KUKA KRL program: EPS_2_251825_SA14_A_20260116064056.src

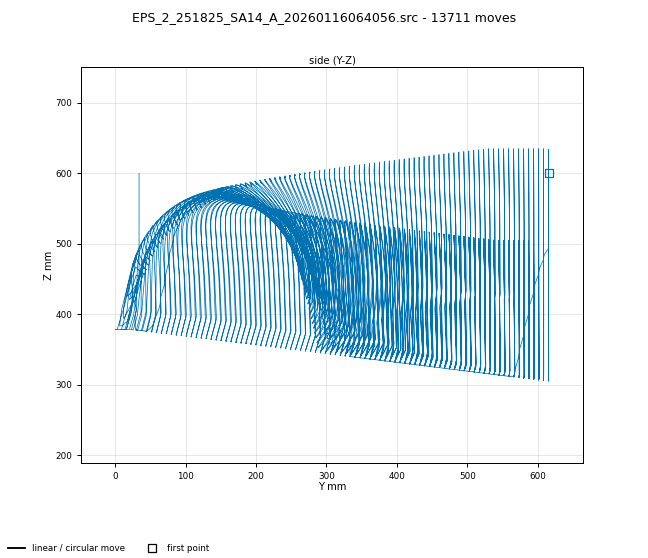
[picture p0: tool path of EPS_2_251825_SA14_A_20260116064056.src, 13711 of 13713 moves have a stored position in this frame; points joined in program order, loops and branches not executed]
&ACCESS RVP
&REL 4
&COMMENT QRS 19112012
&PARAM EDITMASK = *
DEF PART()
EXT BAS (BAS_COMMAND :IN,REAL :IN )
INT I
BAS (#INITMOV,0 )

;KUKA QRS Post kuka4.cps  Date:22-06-2017 !

File_ID=2976

QRS_PRE_INIT()

;Init var - Until changes are made in qrs_pre_init
Outlet_Square_prg=0
Inlet_1_Square_prg=0
Inlet_2_Square_prg=0
Inlet_3_Square_prg=0
Inlet_4_Square_prg=0
Inlet_5_Square_prg=0

Outlet_1={X 0.000, Y 530.070, Z 534.500, B 0.000, E1 0.000 }
Inlet_1={X 0.000, Y 539.340, Z 404.500, B 0.000, E1 92.000 }
Inlet_2={X 0.000, Y 539.340, Z 404.500, B 0.000, E1 262.000 }
Outlet_1_type=201
Inlet_1_type=201
Inlet_2_type=201
;QRS#1=Sidecore dimensions
;QRS#2=200-8" PVC SDR 35
;QRS#3=200-8" PVC SDR 35
;QRS#4=200-8" PVC SDR 35
;QRS#5=
;QRS#6=
;QRS#7=
;QRS#8=
;QRS#9=12-08 PSX
;QRS#10=12-08 PSX
;QRS#11=12-08 PSX
;QRS#12=
;QRS#13=
;QRS#14=
;QRS#15=
;QRS#16=1220x127x914 3'
;QRS#17=EPS Height
;QRS#18=635
;QRS#19=*
;QRS#20= UPDATED VERSION 22-06-2017
;QRS#21=*
Outlet_Square=0100
Inlet_1_Square=0100
Inlet_2_Square=0100
Inlet_3_Square=0
Inlet_4_Square=0
Inlet_5_Square=0
Mill_Square=1
Outlet_Square_Prg=204
Inlet_1_Square_prg=204
Inlet_2_Square_prg=204

QRS_INIT()

$ADVANCE=5

; T1
PTP {E1 173.528,E2 173.528}
PTP {X 0,Y 615.502,A -85,B 0,C 180,E1 173.528,E2 173.528,E3 0,E4 0,E5 0,E6 0}
QRS_SPEED_INIT()
LIN {X 0,Y 615.502,Z 600,A -85,B 0,C 180,E1 173.528,E2 173.528,E3 0,E4 0,E5 0,E6 0} C_VEL
LIN {X 0,Y 615.502,Z 506.059,A -85,B 0,C 180,E1 173.528,E2 173.528} C_VEL
LIN {X 0,Y 615.502,Z 496.473,A -85,B 0,C 180,E1 173.528,E2 173.528} C_VEL
LIN {X 0,Y 615.497,Z 494.64,A -85,B 0,C 180,E1 173.417,E2 173.417} C_VEL
LIN {X 0,Y 615.496,Z 489.786,A -85,B 0,C 180,E1 172.455,E2 172.455} C_VEL
LIN {X 0,Y 615.498,Z 483.532,A -85,B 0,C 180,E1 171.464,E2 171.464} C_VEL
LIN {X 0,Y 615.498,Z 475.676,A -85,B 0,C 180,E1 170.47,E2 170.47} C_VEL
LIN {X 0,Y 615.498,Z 465.867,A -85,B 0,C 180,E1 169.474,E2 169.474} C_VEL
LIN {X 0,Y 615.499,Z 455.563,A -85,B 0,C 180,E1 168.641,E2 168.641} C_VEL
LIN {X 0,Y 615.479,Z 445.348,A -85,B 0,C 180,E1 167.972,E2 167.972} C_VEL
LIN {X 0,Y 615.497,Z 434.148,A -85,B 0,C 180,E1 167.387,E2 167.387} C_VEL
LIN {X 0,Y 615.49,Z 421.521,A -85,B 0,C 180,E1 166.883,E2 166.883} C_VEL
LIN {X 0,Y 615.487,Z 409.783,A -85,B 0,C 180,E1 166.547,E2 166.547} C_VEL
LIN {X 0,Y 615.473,Z 395.857,A -85,B 0,C 180,E1 166.294,E2 166.294} C_VEL
LIN {X 0,Y 615.498,Z 304.699,A -85,B 0,C 180,E1 165.219,E2 165.219} C_VEL
LIN {X 0,Y 615.493,Z 304.685,A -85,B 0,C 180,E1 162.73,E2 162.73} C_VEL
LIN {X 0,Y 615.461,Z 304.691,A -85,B 0,C 180,E1 159.967,E2 159.967} C_VEL
LIN {X 0,Y 615.471,Z 304.695,A -85,B 0,C 180,E1 157.658,E2 157.658} C_VEL
LIN {X 0,Y 615.486,Z 304.691,A -85,B 0,C 180,E1 155.009,E2 155.009} C_VEL
LIN {X 0,Y 615.486,Z 304.687,A -85,B 0,C 180,E1 152.823,E2 152.823} C_VEL
LIN {X 0,Y 615.466,Z 304.688,A -85,B 0,C 180,E1 150.209,E2 150.209} C_VEL
LIN {X 0,Y 615.483,Z 304.7,A -85,B 0,C 180,E1 147.543,E2 147.543} C_VEL
LIN {X 0,Y 615.488,Z 304.693,A -85,B 0,C 180,E1 145.185,E2 145.185} C_VEL
LIN {X 0,Y 615.49,Z 304.683,A -85,B 0,C 180,E1 142.758,E2 142.758} C_VEL
LIN {X 0,Y 615.467,Z 304.694,A -85,B 0,C 180,E1 139.914,E2 139.914} C_VEL
LIN {X 0,Y 615.487,Z 304.698,A -85,B 0,C 180,E1 137.647,E2 137.647} C_VEL
LIN {X 0,Y 615.483,Z 304.686,A -85,B 0,C 180,E1 134.932,E2 134.932} C_VEL
LIN {X 0,Y 615.467,Z 304.692,A -85,B 0,C 180,E1 132.079,E2 132.079} C_VEL
LIN {X 0,Y 615.484,Z 304.698,A -85,B 0,C 180,E1 129.751,E2 129.751} C_VEL
LIN {X 0,Y 615.484,Z 304.685,A -85,B 0,C 180,E1 126.937,E2 126.937} C_VEL
LIN {X 0,Y 615.49,Z 304.682,A -85,B 0,C 180,E1 124.702,E2 124.702} C_VEL
LIN {X 0,Y 615.47,Z 304.689,A -85,B 0,C 180,E1 122.329,E2 122.329} C_VEL
LIN {X 0,Y 615.489,Z 304.699,A -85,B 0,C 180,E1 119.796,E2 119.796} C_VEL
LIN {X 0,Y 615.487,Z 304.684,A -85,B 0,C 180,E1 117.046,E2 117.046} C_VEL
LIN {X 0,Y 615.489,Z 304.683,A -85,B 0,C 180,E1 114.992,E2 114.992} C_VEL
LIN {X 0,Y 615.475,Z 304.693,A -85,B 0,C 180,E1 112.137,E2 112.137} C_VEL
LIN {X 0,Y 615.48,Z 304.69,A -85,B 0,C 180,E1 109.338,E2 109.338} C_VEL
LIN {X 0,Y 615.478,Z 304.686,A -85,B 0,C 180,E1 106.587,E2 106.587} C_VEL
LIN {X 0,Y 615.497,Z 304.7,A -85,B 0,C 180,E1 103.874,E2 103.874} C_VEL
LIN {X 0,Y 615.486,Z 304.683,A -85,B 0,C 180,E1 100.889,E2 100.889} C_VEL
LIN {X 0,Y 615.476,Z 304.688,A -85,B 0,C 180,E1 98.537,E2 98.537} C_VEL
LIN {X 0,Y 615.496,Z 304.7,A -85,B 0,C 180,E1 95.898,E2 95.898} C_VEL
LIN {X 0,Y 615.482,Z 304.686,A -85,B 0,C 180,E1 93.273,E2 93.273} C_VEL
LIN {X 0,Y 615.479,Z 304.686,A -85,B 0,C 180,E1 90.654,E2 90.654} C_VEL
LIN {X 0,Y 615.496,Z 304.7,A -85,B 0,C 180,E1 88.037,E2 88.037} C_VEL
LIN {X 0,Y 615.477,Z 304.688,A -85,B 0,C 180,E1 85.415,E2 85.415} C_VEL
LIN {X 0,Y 615.483,Z 304.685,A -85,B 0,C 180,E1 82.784,E2 82.784} C_VEL
LIN {X 0,Y 615.493,Z 304.699,A -85,B 0,C 180,E1 80.138,E2 80.138} C_VEL
LIN {X 0,Y 615.477,Z 304.687,A -85,B 0,C 180,E1 77.469,E2 77.469} C_VEL
LIN {X 0,Y 615.482,Z 304.686,A -85,B 0,C 180,E1 74.774,E2 74.774} C_VEL
LIN {X 0,Y 615.49,Z 304.698,A -85,B 0,C 180,E1 72.043,E2 72.043} C_VEL
LIN {X 0,Y 615.487,Z 304.682,A -85,B 0,C 180,E1 69.269,E2 69.269} C_VEL
LIN {X 0,Y 615.485,Z 304.695,A -85,B 0,C 180,E1 66.443,E2 66.443} C_VEL
LIN {X 0,Y 615.496,Z 304.699,A -85,B 0,C 180,E1 64.284,E2 64.284} C_VEL
LIN {X 0,Y 615.482,Z 304.683,A -85,B 0,C 180,E1 61.341,E2 61.341} C_VEL
LIN {X 0,Y 615.485,Z 304.686,A -85,B 0,C 180,E1 58.914,E2 58.914} C_VEL
LIN {X 0,Y 615.476,Z 304.694,A -85,B 0,C 180,E1 55.977,E2 55.977} C_VEL
LIN {X 0,Y 615.473,Z 304.687,A -85,B 0,C 180,E1 53.574,E2 53.574} C_VEL
LIN {X 0,Y 615.485,Z 304.686,A -85,B 0,C 180,E1 50.938,E2 50.938} C_VEL
LIN {X 0,Y 615.489,Z 304.697,A -85,B 0,C 180,E1 48.526,E2 48.526} C_VEL
LIN {X 0,Y 615.469,Z 304.69,A -85,B 0,C 180,E1 45.848,E2 45.848} C_VEL
LIN {X 0,Y 615.488,Z 304.685,A -85,B 0,C 180,E1 43.047,E2 43.047} C_VEL
LIN {X 0,Y 615.49,Z 304.697,A -85,B 0,C 180,E1 40.606,E2 40.606} C_VEL
LIN {X 0,Y 615.469,Z 304.692,A -85,B 0,C 180,E1 38.009,E2 38.009} C_VEL
LIN {X 0,Y 615.473,Z 304.686,A -85,B 0,C 180,E1 35.616,E2 35.616} C_VEL
LIN {X 0,Y 615.49,Z 304.683,A -85,B 0,C 180,E1 33.236,E2 33.236} C_VEL
LIN {X 0,Y 615.486,Z 304.691,A -85,B 0,C 180,E1 30.919,E2 30.919} C_VEL
LIN {X 0,Y 615.485,Z 304.699,A -85,B 0,C 180,E1 28.449,E2 28.449} C_VEL
LIN {X 0,Y 615.48,Z 304.684,A -85,B 0,C 180,E1 25.566,E2 25.566} C_VEL
LIN {X 0,Y 615.486,Z 304.696,A -85,B 0,C 180,E1 22.844,E2 22.844} C_VEL
LIN {X 0,Y 615.487,Z 304.702,A -85,B 0,C 180,E1 20.686,E2 20.686} C_VEL
LIN {X 0,Y 615.486,Z 401.466,A -85,B 0,C 180,E1 19.533,E2 19.533} C_VEL
LIN {X 0,Y 615.49,Z 414.153,A -85,B 0,C 180,E1 19.251,E2 19.251} C_VEL
LIN {X 0,Y 615.49,Z 427.253,A -85,B 0,C 180,E1 18.818,E2 18.818} C_VEL
LIN {X 0,Y 615.491,Z 439.133,A -85,B 0,C 180,E1 18.281,E2 18.281} C_VEL
LIN {X 0,Y 615.485,Z 450.58,A -85,B 0,C 180,E1 17.613,E2 17.613} C_VEL
LIN {X 0,Y 615.497,Z 461.144,A -85,B 0,C 180,E1 16.842,E2 16.842} C_VEL
LIN {X 0,Y 615.499,Z 470.075,A -85,B 0,C 180,E1 16.036,E2 16.036} C_VEL
LIN {X 0,Y 615.497,Z 478.904,A -85,B 0,C 180,E1 15.056,E2 15.056} C_VEL
LIN {X 0,Y 615.498,Z 485.954,A -85,B 0,C 180,E1 14.088,E2 14.088} C_VEL
LIN {X 0,Y 615.499,Z 491.179,A -85,B 0,C 180,E1 13.201,E2 13.201} C_VEL
LIN {X 0,Y 615.495,Z 495.923,A -85,B 0,C 180,E1 12.195,E2 12.195} C_VEL
LIN {X 0,Y 615.496,Z 499.511,A -85,B 0,C 180,E1 11.193,E2 11.193} C_VEL
LIN {X 0,Y 615.497,Z 501.344,A -85,B 0,C 180,E1 10.526,E2 10.526} C_VEL
LIN {X 0,Y 615.495,Z 502.702,A -85,B 0,C 180,E1 9.862,E2 9.862} C_VEL
LIN {X 0,Y 615.496,Z 504.225,A -85,B 0,C 180,E1 8.536,E2 8.536} C_VEL
LIN {X 0,Y 615.495,Z 504.376,A -85,B 0,C 180,E1 7.875,E2 7.875} C_VEL
LIN {X 0,Y 615.497,Z 503.473,A -85,B 0,C 180,E1 6.556,E2 6.556} C_VEL
LIN {X 0,Y 615.499,Z 502.449,A -85,B 0,C 180,E1 5.898,E2 5.898} C_VEL
LIN {X 0,Y 615.495,Z 500.977,A -85,B 0,C 180,E1 5.241,E2 5.241} C_VEL
LIN {X 0,Y 615.496,Z 497.999,A -85,B 0,C 180,E1 4.256,E2 4.256} C_VEL
LIN {X 0,Y 615.496,Z 493.997,A -85,B 0,C 180,E1 3.273,E2 3.273} C_VEL
LIN {X 0,Y 615.496,Z 487.85,A -85,B 0,C 180,E1 2.126,E2 2.126} C_VEL
LIN {X 0,Y 615.498,Z 481.175,A -85,B 0,C 180,E1 1.145,E2 1.145} C_VEL
LIN {X 0,Y 615.498,Z 472.909,A -85,B 0,C 180,E1 0.163,E2 0.163} C_VEL
LIN {X 0,Y 615.498,Z 464.406,A -85,B 0,C 180,E1 -0.655,E2 -0.655} C_VEL
LIN {X 0,Y 615.493,Z 453.986,A -85,B 0,C 180,E1 -1.472,E2 -1.472} C_VEL
LIN {X 0,Y 615.476,Z 443.668,A -85,B 0,C 180,E1 -2.127,E2 -2.127} C_VEL
LIN {X 0,Y 615.49,Z 432.239,A -85,B 0,C 180,E1 -2.7,E2 -2.7} C_VEL
LIN {X 0,Y 615.452,Z 420.503,A -85,B 0,C 180,E1 -3.151,E2 -3.151} C_VEL
LIN {X 0,Y 615.434,Z 408.729,A -85,B 0,C 180,E1 -3.478,E2 -3.478} C_VEL
LIN {X 0,Y 615.432,Z 396.068,A -85,B 0,C 180,E1 -3.704,E2 -3.704} C_VEL
LIN {X 0,Y 615.484,Z 304.701,A -85,B 0,C 180,E1 -4.79,E2 -4.79} C_VEL
LIN {X 0,Y 615.438,Z 304.698,A -85,B 0,C 180,E1 -7.217,E2 -7.217} C_VEL
LIN {X 0,Y 615.432,Z 304.699,A -85,B 0,C 180,E1 -9.2,E2 -9.2} C_VEL
LIN {X 0,Y 615.431,Z 304.699,A -85,B 0,C 180,E1 -11.194,E2 -11.194} C_VEL
LIN {X 0,Y 615.426,Z 304.699,A -85,B 0,C 180,E1 -13.203,E2 -13.203} C_VEL
LIN {X 0,Y 615.421,Z 304.699,A -85,B 0,C 180,E1 -15.228,E2 -15.228} C_VEL
LIN {X 0,Y 615.415,Z 304.7,A -85,B 0,C 180,E1 -17.273,E2 -17.273} C_VEL
LIN {X 0,Y 615.411,Z 304.7,A -85,B 0,C 180,E1 -19.341,E2 -19.341} C_VEL
LIN {X 0,Y 615.412,Z 304.7,A -85,B 0,C 180,E1 -21.435,E2 -21.435} C_VEL
LIN {X 0,Y 615.456,Z 304.7,A -85,B 0,C 180,E1 -24.001,E2 -24.001} C_VEL
LIN {X 0,Y 615.486,Z 304.696,A -85,B 0,C 180,E1 -26.445,E2 -26.445} C_VEL
LIN {X 0,Y 615.456,Z 304.696,A -85,B 0,C 180,E1 -28.66,E2 -28.66} C_VEL
LIN {X 0,Y 615.428,Z 304.696,A -85,B 0,C 180,E1 -31.076,E2 -31.076} C_VEL
LIN {X 0,Y 615.428,Z 304.697,A -85,B 0,C 180,E1 -33.24,E2 -33.24} C_VEL
LIN {X 0,Y 615.471,Z 304.699,A -85,B 0,C 180,E1 -35.831,E2 -35.831} C_VEL
LIN {X 0,Y 615.49,Z 304.699,A -85,B 0,C 180,E1 -38.069,E2 -38.069} C_VEL
LIN {X 0,Y 615.46,Z 304.691,A -85,B 0,C 180,E1 -40.609,E2 -40.609} C_VEL
LIN {X 0,Y 615.441,Z 304.694,A -85,B 0,C 180,E1 -43.042,E2 -43.042} C_VEL
LIN {X 0,Y 615.443,Z 304.694,A -85,B 0,C 180,E1 -45.073,E2 -45.073} C_VEL
LIN {X 0,Y 615.483,Z 304.699,A -85,B 0,C 180,E1 -47.646,E2 -47.646} C_VEL
LIN {X 0,Y 615.493,Z 304.686,A -85,B 0,C 180,E1 -50.25,E2 -50.25} C_VEL
LIN {X 0,Y 615.454,Z 304.69,A -85,B 0,C 180,E1 -52.755,E2 -52.755} C_VEL
LIN {X 0,Y 615.469,Z 304.697,A -85,B 0,C 180,E1 -55.302,E2 -55.302} C_VEL
LIN {X 0,Y 615.482,Z 304.685,A -85,B 0,C 180,E1 -58.314,E2 -58.314} C_VEL
LIN {X 0,Y 615.465,Z 304.688,A -85,B 0,C 180,E1 -60.592,E2 -60.592} C_VEL
LIN {X 0,Y 615.464,Z 304.693,A -85,B 0,C 180,E1 -62.96,E2 -62.96} C_VEL
LIN {X 0,Y 615.467,Z 304.836,A -85,B 0,C 180,E1 -64.578,E2 -64.578} C_VEL
LIN {X 0,Y 615.488,Z 329.133,A -85,B 0,C 180,E1 -67.281,E2 -67.281} C_VEL
LIN {X 0,Y 615.496,Z 355.374,A -85,B 0,C 180,E1 -70.141,E2 -70.141} C_VEL
LIN {X 0,Y 615.493,Z 382.737,A -85,B 0,C 180,E1 -73.072,E2 -73.072} C_VEL
LIN {X 0,Y 615.499,Z 411.083,A -85,B 0,C 180,E1 -76.064,E2 -76.064} C_VEL
LIN {X 0,Y 615.498,Z 421.301,A -85,B 0,C 180,E1 -77.114,E2 -77.114} C_VEL
LIN {X 0,Y 615.479,Z 530.821,A -85,B 0,C 180,E1 -78.41,E2 -78.41} C_VEL
LIN {X 0,Y 615.478,Z 543.339,A -85,B 0,C 180,E1 -78.681,E2 -78.681} C_VEL
LIN {X 0,Y 615.491,Z 556.57,A -85,B 0,C 180,E1 -79.111,E2 -79.111} C_VEL
LIN {X 0,Y 615.478,Z 568.475,A -85,B 0,C 180,E1 -79.639,E2 -79.639} C_VEL
LIN {X 0,Y 615.487,Z 579.992,A -85,B 0,C 180,E1 -80.304,E2 -80.304} C_VEL
LIN {X 0,Y 615.499,Z 590.339,A -85,B 0,C 180,E1 -81.05,E2 -81.05} C_VEL
LIN {X 0,Y 615.497,Z 598.81,A -85,B 0,C 180,E1 -81.794,E2 -81.794} C_VEL
LIN {X 0,Y 615.498,Z 606.605,A -85,B 0,C 180,E1 -82.619,E2 -82.619} C_VEL
LIN {X 0,Y 615.496,Z 614.202,A -85,B 0,C 180,E1 -83.608,E2 -83.608} C_VEL
LIN {X 0,Y 615.498,Z 621.204,A -85,B 0,C 180,E1 -84.759,E2 -84.759} C_VEL
LIN {X 0,Y 615.493,Z 625.851,A -85,B 0,C 180,E1 -85.743,E2 -85.743} C_VEL
LIN {X 0,Y 615.495,Z 629.398,A -85,B 0,C 180,E1 -86.727,E2 -86.727} C_VEL
LIN {X 0,Y 615.497,Z 631.233,A -85,B 0,C 180,E1 -87.382,E2 -87.382} C_VEL
LIN {X 0,Y 615.497,Z 632.608,A -85,B 0,C 180,E1 -88.037,E2 -88.037} C_VEL
LIN {X 0,Y 615.496,Z 634.173,A -85,B 0,C 180,E1 -89.346,E2 -89.346} C_VEL
LIN {X 0,Y 615.494,Z 634.389,A -85,B 0,C 180,E1 -90,E2 -90} C_VEL
LIN {X 0,Y 615.496,Z 633.58,A -85,B 0,C 180,E1 -91.308,E2 -91.308} C_VEL
LIN {X 0,Y 615.497,Z 632.608,A -85,B 0,C 180,E1 -91.963,E2 -91.963} C_VEL
LIN {X 0,Y 615.497,Z 631.233,A -85,B 0,C 180,E1 -92.618,E2 -92.618} C_VEL
LIN {X 0,Y 615.496,Z 628.35,A -85,B 0,C 180,E1 -93.601,E2 -93.601} C_VEL
LIN {X 0,Y 615.498,Z 624.442,A -85,B 0,C 180,E1 -94.584,E2 -94.584} C_VEL
LIN {X 0,Y 615.499,Z 619.405,A -85,B 0,C 180,E1 -95.57,E2 -95.57} C_VEL
LIN {X 0,Y 615.497,Z 612.87,A -85,B 0,C 180,E1 -96.583,E2 -96.583} C_VEL
LIN {X 0,Y 615.497,Z 605.134,A -85,B 0,C 180,E1 -97.545,E2 -97.545} C_VEL
LIN {X 0,Y 615.498,Z 597.045,A -85,B 0,C 180,E1 -98.371,E2 -98.371} C_VEL
LIN {X 0,Y 615.499,Z 587.168,A -85,B 0,C 180,E1 -99.199,E2 -99.199} C_VEL
LIN {X 0,Y 615.488,Z 575.982,A -85,B 0,C 180,E1 -99.945,E2 -99.945} C_VEL
LIN {X 0,Y 615.481,Z 565.024,A -85,B 0,C 180,E1 -100.527,E2 -100.527} C_VEL
LIN {X 0,Y 615.49,Z 552.45,A -85,B 0,C 180,E1 -101.041,E2 -101.041} C_VEL
LIN {X 0,Y 615.477,Z 540.068,A -85,B 0,C 180,E1 -101.402,E2 -101.402} C_VEL
LIN {X 0,Y 615.481,Z 526.47,A -85,B 0,C 180,E1 -101.652,E2 -101.652} C_VEL
LIN {X 0,Y 615.499,Z 420.901,A -85,B 0,C 180,E1 -102.907,E2 -102.907} C_VEL
LIN {X 0,Y 615.486,Z 393.999,A -85,B 0,C 180,E1 -105.735,E2 -105.735} C_VEL
LIN {X 0,Y 615.477,Z 368.567,A -85,B 0,C 180,E1 -108.441,E2 -108.441} C_VEL
LIN {X 0,Y 615.498,Z 344.101,A -85,B 0,C 180,E1 -111.081,E2 -111.081} C_VEL
LIN {X 0,Y 615.487,Z 318.499,A -85,B 0,C 180,E1 -113.895,E2 -113.895} C_VEL
LIN {X 0,Y 615.468,Z 304.687,A -85,B 0,C 180,E1 -115.458,E2 -115.458} C_VEL
LIN {X 0,Y 615.493,Z 304.699,A -85,B 0,C 180,E1 -118.451,E2 -118.451} C_VEL
LIN {X 0,Y 615.457,Z 304.693,A -85,B 0,C 180,E1 -121.081,E2 -121.081} C_VEL
LIN {X 0,Y 615.471,Z 304.687,A -85,B 0,C 180,E1 -123.531,E2 -123.531} C_VEL
LIN {X 0,Y 615.483,Z 304.701,A -85,B 0,C 180,E1 -126.425,E2 -126.425} C_VEL
LIN {X 0,Y 615.449,Z 304.692,A -85,B 0,C 180,E1 -129.057,E2 -129.057} C_VEL
LIN {X 0,Y 615.467,Z 304.689,A -85,B 0,C 180,E1 -131.476,E2 -131.476} C_VEL
LIN {X 0,Y 615.496,Z 304.7,A -85,B 0,C 180,E1 -134.149,E2 -134.149} C_VEL
LIN {X 0,Y 615.442,Z 304.695,A -85,B 0,C 180,E1 -136.751,E2 -136.751} C_VEL
LIN {X 0,Y 615.437,Z 304.695,A -85,B 0,C 180,E1 -138.911,E2 -138.911} C_VEL
LIN {X 0,Y 615.439,Z 304.694,A -85,B 0,C 180,E1 -141.092,E2 -141.092} C_VEL
LIN {X 0,Y 615.479,Z 304.693,A -85,B 0,C 180,E1 -143.574,E2 -143.574} C_VEL
LIN {X 0,Y 615.436,Z 304.698,A -85,B 0,C 180,E1 -146.473,E2 -146.473} C_VEL
LIN {X 0,Y 615.443,Z 304.699,A -85,B 0,C 180,E1 -148.312,E2 -148.312} C_VEL
LIN {X 0,Y 615.423,Z 304.698,A -85,B 0,C 180,E1 -150.59,E2 -150.59} C_VEL
LIN {X 0,Y 615.424,Z 304.698,A -85,B 0,C 180,E1 -152.967,E2 -152.967} C_VEL
LIN {X 0,Y 615.482,Z 304.702,A -85,B 0,C 180,E1 -155.727,E2 -155.727} C_VEL
LIN {X 0,Y 615.462,Z 304.701,A -85,B 0,C 180,E1 -157.862,E2 -157.862} C_VEL
LIN {X 0,Y 615.448,Z 304.699,A -85,B 0,C 180,E1 -159.966,E2 -159.966} C_VEL
LIN {X 0,Y 615.441,Z 304.698,A -85,B 0,C 180,E1 -162.041,E2 -162.041} C_VEL
LIN {X 0,Y 615.436,Z 304.697,A -85,B 0,C 180,E1 -164.093,E2 -164.093} C_VEL
LIN {X 0,Y 615.435,Z 304.697,A -85,B 0,C 180,E1 -166.124,E2 -166.124} C_VEL
LIN {X 0,Y 615.435,Z 304.696,A -85,B 0,C 180,E1 -168.138,E2 -168.138} C_VEL
LIN {X 0,Y 615.482,Z 304.701,A -85,B 0,C 180,E1 -169.299,E2 -169.299} C_VEL
LIN {X 0,Y 615.427,Z 401.605,A -85,B 0,C 180,E1 -170.468,E2 -170.468} C_VEL
LIN {X 0,Y 615.437,Z 414.547,A -85,B 0,C 180,E1 -170.759,E2 -170.759} C_VEL
LIN {X 0,Y 615.471,Z 427.039,A -85,B 0,C 180,E1 -171.173,E2 -171.173} C_VEL
LIN {X 0,Y 615.487,Z 438.981,A -85,B 0,C 180,E1 -171.711,E2 -171.711} C_VEL
LIN {X 0,Y 615.486,Z 450.346,A -85,B 0,C 180,E1 -172.372,E2 -172.372} C_VEL
LIN {X 0,Y 615.498,Z 460.41,A -85,B 0,C 180,E1 -173.1,E2 -173.1} C_VEL
LIN {X 0,Y 615.497,Z 469.813,A -85,B 0,C 180,E1 -173.937,E2 -173.937} C_VEL
LIN {X 0,Y 615.496,Z 478.73,A -85,B 0,C 180,E1 -174.923,E2 -174.923} C_VEL
LIN {X 0,Y 615.497,Z 485.922,A -85,B 0,C 180,E1 -175.907,E2 -175.907} C_VEL
LIN {X 0,Y 615.497,Z 490.782,A -85,B 0,C 180,E1 -176.727,E2 -176.727} C_VEL
LIN {X 0,Y 615.496,Z 495.51,A -85,B 0,C 180,E1 -177.709,E2 -177.709} C_VEL
LIN {X 0,Y 615.497,Z 499.139,A -85,B 0,C 180,E1 -178.691,E2 -178.691} C_VEL
LIN {X 0,Y 615.495,Z 501.016,A -85,B 0,C 180,E1 -179.345,E2 -179.345} C_VEL
LIN {X 0,Y 615.494,Z 502.471,A -85,B 0,C 180,E1 -180,E2 -180} C_VEL
LIN {X 0,Y 615.495,Z 504.115,A -85,B 0,C 180,E1 -181.308,E2 -181.308} C_VEL
LIN {X 0,Y 615.497,Z 504.374,A -85,B 0,C 180,E1 -181.963,E2 -181.963} C_VEL
LIN {X 0,Y 615.497,Z 504.231,A -85,B 0,C 180,E1 -182.618,E2 -182.618} C_VEL
LIN {X 0,Y 615.496,Z 502.741,A -85,B 0,C 180,E1 -183.928,E2 -183.928} C_VEL
LIN {X 0,Y 615.499,Z 501.416,A -85,B 0,C 180,E1 -184.584,E2 -184.584} C_VEL
LIN {X 0,Y 615.496,Z 498.594,A -85,B 0,C 180,E1 -185.569,E2 -185.569} C_VEL
LIN {X 0,Y 615.497,Z 494.64,A -85,B 0,C 180,E1 -186.583,E2 -186.583} C_VEL
LIN {X 0,Y 614.81,Z 492.425,A -85,B 0,C 180,E1 -187.083,E2 -187.083} C_VEL
LIN {X 0,Y 611.93,Z 488.432,A -85,B 0,C 180,E1 -187.883,E2 -187.883} C_VEL
LIN {X 0,Y 609.08,Z 483.559,A -85,B 0,C 180,E1 -188.659,E2 -188.659} C_VEL
LIN {X 0,Y 608.468,Z 480.16,A -85,B 0,C 180,E1 -189.119,E2 -189.119} C_VEL
LIN {X 0,Y 608.481,Z 471.123,A -85,B 0,C 180,E1 -190.145,E2 -190.145} C_VEL
LIN {X 0,Y 608.48,Z 462.308,A -85,B 0,C 180,E1 -190.96,E2 -190.96} C_VEL
LIN {X 0,Y 608.491,Z 451.844,A -85,B 0,C 180,E1 -191.745,E2 -191.745} C_VEL
LIN {X 0,Y 608.49,Z 440.568,A -85,B 0,C 180,E1 -192.422,E2 -192.422} C_VEL
LIN {X 0,Y 608.513,Z 429.877,A -85,B 0,C 180,E1 -192.93,E2 -192.93} C_VEL
LIN {X 0,Y 608.52,Z 418.273,A -85,B 0,C 180,E1 -193.355,E2 -193.355} C_VEL
LIN {X 0,Y 608.544,Z 404.945,A -85,B 0,C 180,E1 -193.695,E2 -193.695} C_VEL
LIN {X 0,Y 608.532,Z 388.171,A -85,B 0,C 180,E1 -193.935,E2 -193.935} C_VEL
LIN {X 0,Y 608.491,Z 305.69,A -85,B 0,C 180,E1 -194.912,E2 -194.912} C_VEL
LIN {X 0,Y 608.45,Z 305.688,A -85,B 0,C 180,E1 -197.476,E2 -197.476} C_VEL
LIN {X 0,Y 608.445,Z 305.688,A -85,B 0,C 180,E1 -199.57,E2 -199.57} C_VEL
LIN {X 0,Y 608.464,Z 305.686,A -85,B 0,C 180,E1 -201.691,E2 -201.691} C_VEL
LIN {X 0,Y 608.445,Z 305.698,A -85,B 0,C 180,E1 -204.571,E2 -204.571} C_VEL
LIN {X 0,Y 608.48,Z 305.686,A -85,B 0,C 180,E1 -207.207,E2 -207.207} C_VEL
LIN {X 0,Y 608.45,Z 305.689,A -85,B 0,C 180,E1 -209.968,E2 -209.968} C_VEL
LIN {X 0,Y 608.459,Z 305.692,A -85,B 0,C 180,E1 -212.879,E2 -212.879} C_VEL
LIN {X 0,Y 608.437,Z 305.69,A -85,B 0,C 180,E1 -215.278,E2 -215.278} C_VEL
LIN {X 0,Y 608.457,Z 305.687,A -85,B 0,C 180,E1 -217.747,E2 -217.747} C_VEL
LIN {X 0,Y 608.444,Z 305.696,A -85,B 0,C 180,E1 -220.328,E2 -220.328} C_VEL
LIN {X 0,Y 608.483,Z 305.684,A -85,B 0,C 180,E1 -223.31,E2 -223.31} C_VEL
LIN {X 0,Y 608.458,Z 305.692,A -85,B 0,C 180,E1 -226.129,E2 -226.129} C_VEL
LIN {X 0,Y 608.456,Z 305.691,A -85,B 0,C 180,E1 -228.823,E2 -228.823} C_VEL
LIN {X 0,Y 608.466,Z 305.686,A -85,B 0,C 180,E1 -231.412,E2 -231.412} C_VEL
LIN {X 0,Y 608.444,Z 305.692,A -85,B 0,C 180,E1 -233.954,E2 -233.954} C_VEL
LIN {X 0,Y 608.463,Z 305.697,A -85,B 0,C 180,E1 -236.329,E2 -236.329} C_VEL
LIN {X 0,Y 608.476,Z 305.688,A -85,B 0,C 180,E1 -238.727,E2 -238.727} C_VEL
LIN {X 0,Y 608.466,Z 305.686,A -85,B 0,C 180,E1 -241.381,E2 -241.381} C_VEL
LIN {X 0,Y 608.478,Z 305.695,A -85,B 0,C 180,E1 -244.277,E2 -244.277} C_VEL
LIN {X 0,Y 608.451,Z 305.689,A -85,B 0,C 180,E1 -246.876,E2 -246.876} C_VEL
LIN {X 0,Y 608.456,Z 305.69,A -85,B 0,C 180,E1 -249.726,E2 -249.726} C_VEL
LIN {X 0,Y 608.45,Z 305.692,A -85,B 0,C 180,E1 -252.523,E2 -252.523} C_VEL
LIN {X 0,Y 608.468,Z 305.686,A -85,B 0,C 180,E1 -255.279,E2 -255.279} C_VEL
LIN {X 0,Y 608.46,Z 305.695,A -85,B 0,C 180,E1 -258,E2 -258} C_VEL
LIN {X 0,Y 608.467,Z 305.687,A -85,B 0,C 180,E1 -260.694,E2 -260.694} C_VEL
LIN {X 0,Y 608.455,Z 305.688,A -85,B 0,C 180,E1 -263.384,E2 -263.384} C_VEL
LIN {X 0,Y 608.454,Z 305.698,A -85,B 0,C 180,E1 -266.026,E2 -266.026} C_VEL
LIN {X 0,Y 608.466,Z 305.687,A -85,B 0,C 180,E1 -268.676,E2 -268.676} C_VEL
LIN {X 0,Y 608.465,Z 305.687,A -85,B 0,C 180,E1 -271.324,E2 -271.324} C_VEL
LIN {X 0,Y 608.455,Z 305.698,A -85,B 0,C 180,E1 -273.974,E2 -273.974} C_VEL
LIN {X 0,Y 608.458,Z 305.688,A -85,B 0,C 180,E1 -276.633,E2 -276.633} C_VEL
LIN {X 0,Y 608.466,Z 305.687,A -85,B 0,C 180,E1 -279.306,E2 -279.306} C_VEL
LIN {X 0,Y 608.46,Z 305.695,A -85,B 0,C 180,E1 -282,E2 -282} C_VEL
LIN {X 0,Y 608.468,Z 305.686,A -85,B 0,C 180,E1 -284.721,E2 -284.721} C_VEL
LIN {X 0,Y 608.45,Z 305.692,A -85,B 0,C 180,E1 -287.477,E2 -287.477} C_VEL
LIN {X 0,Y 608.458,Z 305.69,A -85,B 0,C 180,E1 -290.275,E2 -290.275} C_VEL
LIN {X 0,Y 608.45,Z 305.689,A -85,B 0,C 180,E1 -293.124,E2 -293.124} C_VEL
LIN {X 0,Y 608.476,Z 305.695,A -85,B 0,C 180,E1 -295.723,E2 -295.723} C_VEL
LIN {X 0,Y 608.442,Z 305.691,A -85,B 0,C 180,E1 -298.267,E2 -298.267} C_VEL
LIN {X 0,Y 608.468,Z 305.686,A -85,B 0,C 180,E1 -300.545,E2 -300.545} C_VEL
LIN {X 0,Y 608.451,Z 305.688,A -85,B 0,C 180,E1 -302.88,E2 -302.88} C_VEL
LIN {X 0,Y 608.454,Z 305.691,A -85,B 0,C 180,E1 -305.277,E2 -305.277} C_VEL
LIN {X 0,Y 608.462,Z 305.695,A -85,B 0,C 180,E1 -307.747,E2 -307.747} C_VEL
LIN {X 0,Y 608.44,Z 305.69,A -85,B 0,C 180,E1 -310.328,E2 -310.328} C_VEL
LIN {X 0,Y 608.472,Z 305.691,A -85,B 0,C 180,E1 -313.31,E2 -313.31} C_VEL
LIN {X 0,Y 608.46,Z 305.689,A -85,B 0,C 180,E1 -316.13,E2 -316.13} C_VEL
LIN {X 0,Y 608.453,Z 305.688,A -85,B 0,C 180,E1 -318.824,E2 -318.824} C_VEL
LIN {X 0,Y 608.457,Z 305.693,A -85,B 0,C 180,E1 -321.762,E2 -321.762} C_VEL
LIN {X 0,Y 608.443,Z 305.692,A -85,B 0,C 180,E1 -323.956,E2 -323.956} C_VEL
LIN {X 0,Y 608.444,Z 305.688,A -85,B 0,C 180,E1 -326.329,E2 -326.329} C_VEL
LIN {X 0,Y 608.449,Z 305.689,A -85,B 0,C 180,E1 -328.733,E2 -328.733} C_VEL
LIN {X 0,Y 608.473,Z 305.695,A -85,B 0,C 180,E1 -331.381,E2 -331.381} C_VEL
LIN {X 0,Y 608.435,Z 305.691,A -85,B 0,C 180,E1 -333.964,E2 -333.964} C_VEL
LIN {X 0,Y 608.452,Z 305.688,A -85,B 0,C 180,E1 -336.155,E2 -336.155} C_VEL
LIN {X 0,Y 608.461,Z 305.692,A -85,B 0,C 180,E1 -339.019,E2 -339.019} C_VEL
LIN {X 0,Y 608.487,Z 305.821,A -85,B 0,C 180,E1 -339.179,E2 -339.179} C_VEL
LIN {X 0,Y 608.535,Z 401.017,A -85,B 0,C 180,E1 -340.323,E2 -340.323} C_VEL
LIN {X 0,Y 608.538,Z 414.694,A -85,B 0,C 180,E1 -340.63,E2 -340.63} C_VEL
LIN {X 0,Y 608.535,Z 427.121,A -85,B 0,C 180,E1 -341.046,E2 -341.046} C_VEL
LIN {X 0,Y 608.496,Z 438.995,A -85,B 0,C 180,E1 -341.584,E2 -341.584} C_VEL
LIN {X 0,Y 608.478,Z 450.622,A -85,B 0,C 180,E1 -342.264,E2 -342.264} C_VEL
LIN {X 0,Y 608.485,Z 461.269,A -85,B 0,C 180,E1 -343.044,E2 -343.044} C_VEL
LIN {X 0,Y 608.461,Z 470.747,A -85,B 0,C 180,E1 -343.907,E2 -343.907} C_VEL
LIN {X 0,Y 608.446,Z 479.89,A -85,B 0,C 180,E1 -344.937,E2 -344.937} C_VEL
LIN {X 0,Y 608.445,Z 487.358,A -85,B 0,C 180,E1 -345.994,E2 -345.994} C_VEL
LIN {X 0,Y 608.433,Z 492.919,A -85,B 0,C 180,E1 -346.983,E2 -346.983} C_VEL
LIN {X 0,Y 608.445,Z 497.413,A -85,B 0,C 180,E1 -348,E2 -348} C_VEL
LIN {X 0,Y 608.423,Z 500.937,A -85,B 0,C 180,E1 -349.07,E2 -349.07} C_VEL
LIN {X 0,Y 608.432,Z 503.141,A -85,B 0,C 180,E1 -350.023,E2 -350.023} C_VEL
LIN {X 0,Y 608.42,Z 504.77,A -85,B 0,C 180,E1 -351.364,E2 -351.364} C_VEL
LIN {X 0,Y 608.42,Z 505,A -85,B 0,C 180,E1 -352.033,E2 -352.033} C_VEL
LIN {X 0,Y 608.449,Z 504.185,A -85,B 0,C 180,E1 -353.367,E2 -353.367} C_VEL
LIN {X 0,Y 608.435,Z 503.198,A -85,B 0,C 180,E1 -354.033,E2 -354.033} C_VEL
LIN {X 0,Y 608.438,Z 501.796,A -85,B 0,C 180,E1 -354.698,E2 -354.698} C_VEL
LIN {X 0,Y 608.441,Z 498.871,A -85,B 0,C 180,E1 -355.694,E2 -355.694} C_VEL
LIN {X 0,Y 608.43,Z 494.92,A -85,B 0,C 180,E1 -356.689,E2 -356.689} C_VEL
LIN {X 0,Y 608.459,Z 489.842,A -85,B 0,C 180,E1 -357.683,E2 -357.683} C_VEL
LIN {X 0,Y 608.451,Z 483.481,A -85,B 0,C 180,E1 -358.677,E2 -358.677} C_VEL
LIN {X 0,Y 608.468,Z 475.554,A -85,B 0,C 180,E1 -359.669,E2 -359.669} C_VEL
LIN {X 0,Y 608.492,Z 465.737,A -85,B 0,C 180,E1 -360.662,E2 -360.662} C_VEL
LIN {X 0,Y 608.481,Z 455.491,A -85,B 0,C 180,E1 -361.489,E2 -361.489} C_VEL
LIN {X 0,Y 608.492,Z 444.009,A -85,B 0,C 180,E1 -362.234,E2 -362.234} C_VEL
LIN {X 0,Y 608.523,Z 432.595,A -85,B 0,C 180,E1 -362.814,E2 -362.814} C_VEL
LIN {X 0,Y 608.507,Z 420.901,A -85,B 0,C 180,E1 -363.269,E2 -363.269} C_VEL
LIN {X 0,Y 608.483,Z 407.453,A -85,B 0,C 180,E1 -363.642,E2 -363.642} C_VEL
LIN {X 0,Y 608.489,Z 393.709,A -85,B 0,C 180,E1 -363.87,E2 -363.87} C_VEL
LIN {X 0,Y 608.519,Z 306.051,A -85,B 0,C 180,E1 -364.907,E2 -364.907} C_VEL
LIN {X 0,Y 608.444,Z 305.696,A -85,B 0,C 180,E1 -364.929,E2 -364.929} C_VEL
LIN {X 0,Y 608.415,Z 305.694,A -85,B 0,C 180,E1 -367.3,E2 -367.3} C_VEL
LIN {X 0,Y 608.42,Z 305.693,A -85,B 0,C 180,E1 -369.307,E2 -369.307} C_VEL
LIN {X 0,Y 608.41,Z 305.694,A -85,B 0,C 180,E1 -371.325,E2 -371.325} C_VEL
LIN {X 0,Y 608.409,Z 305.693,A -85,B 0,C 180,E1 -373.358,E2 -373.358} C_VEL
LIN {X 0,Y 608.43,Z 305.695,A -85,B 0,C 180,E1 -376.095,E2 -376.095} C_VEL
LIN {X 0,Y 608.434,Z 305.693,A -85,B 0,C 180,E1 -378.871,E2 -378.871} C_VEL
LIN {X 0,Y 608.418,Z 305.693,A -85,B 0,C 180,E1 -380.983,E2 -380.983} C_VEL
LIN {X 0,Y 608.401,Z 305.694,A -85,B 0,C 180,E1 -383.126,E2 -383.126} C_VEL
LIN {X 0,Y 608.426,Z 305.693,A -85,B 0,C 180,E1 -385.711,E2 -385.711} C_VEL
LIN {X 0,Y 608.432,Z 305.694,A -85,B 0,C 180,E1 -388.612,E2 -388.612} C_VEL
LIN {X 0,Y 608.41,Z 305.693,A -85,B 0,C 180,E1 -391.32,E2 -391.32} C_VEL
LIN {X 0,Y 608.429,Z 305.695,A -85,B 0,C 180,E1 -393.728,E2 -393.728} C_VEL
LIN {X 0,Y 608.446,Z 305.698,A -85,B 0,C 180,E1 -396.093,E2 -396.093} C_VEL
LIN {X 0,Y 608.415,Z 305.694,A -85,B 0,C 180,E1 -398.592,E2 -398.592} C_VEL
LIN {X 0,Y 608.41,Z 305.693,A -85,B 0,C 180,E1 -401.181,E2 -401.181} C_VEL
LIN {X 0,Y 608.468,Z 305.696,A -85,B 0,C 180,E1 -403.87,E2 -403.87} C_VEL
LIN {X 0,Y 608.444,Z 305.689,A -85,B 0,C 180,E1 -406.694,E2 -406.694} C_VEL
LIN {X 0,Y 608.422,Z 305.691,A -85,B 0,C 180,E1 -408.82,E2 -408.82} C_VEL
LIN {X 0,Y 608.469,Z 305.695,A -85,B 0,C 180,E1 -411.76,E2 -411.76} C_VEL
LIN {X 0,Y 608.431,Z 305.69,A -85,B 0,C 180,E1 -414.721,E2 -414.721} C_VEL
LIN {X 0,Y 608.466,Z 305.695,A -85,B 0,C 180,E1 -417.477,E2 -417.477} C_VEL
LIN {X 0,Y 608.48,Z 305.685,A -85,B 0,C 180,E1 -420.221,E2 -420.221} C_VEL
LIN {X 0,Y 608.44,Z 305.691,A -85,B 0,C 180,E1 -422.8,E2 -422.8} C_VEL
LIN {X 0,Y 608.505,Z 305.877,A -85,B 0,C 180,E1 -424.384,E2 -424.384} C_VEL
LIN {X 0,Y 608.672,Z 319.526,A -85,B 0,C 180,E1 -425.936,E2 -425.936} C_VEL
LIN {X 0,Y 608.62,Z 344.099,A -85,B 0,C 180,E1 -428.669,E2 -428.669} C_VEL
LIN {X 0,Y 608.571,Z 368.97,A -85,B 0,C 180,E1 -431.386,E2 -431.386} C_VEL
LIN {X 0,Y 608.532,Z 395.643,A -85,B 0,C 180,E1 -434.252,E2 -434.252} C_VEL
LIN {X 0,Y 608.528,Z 421.336,A -85,B 0,C 180,E1 -436.963,E2 -436.963} C_VEL
LIN {X 0,Y 608.538,Z 530.936,A -85,B 0,C 180,E1 -438.276,E2 -438.276} C_VEL
LIN {X 0,Y 608.514,Z 544.209,A -85,B 0,C 180,E1 -438.571,E2 -438.571} C_VEL
LIN {X 0,Y 608.517,Z 556.597,A -85,B 0,C 180,E1 -438.981,E2 -438.981} C_VEL
LIN {X 0,Y 608.498,Z 568.631,A -85,B 0,C 180,E1 -439.519,E2 -439.519} C_VEL
LIN {X 0,Y 608.48,Z 580.194,A -85,B 0,C 180,E1 -440.191,E2 -440.191} C_VEL
LIN {X 0,Y 608.485,Z 590.591,A -85,B 0,C 180,E1 -440.946,E2 -440.946} C_VEL
LIN {X 0,Y 608.475,Z 599.11,A -85,B 0,C 180,E1 -441.699,E2 -441.699} C_VEL
LIN {X 0,Y 608.471,Z 606.959,A -85,B 0,C 180,E1 -442.534,E2 -442.534} C_VEL
LIN {X 0,Y 608.461,Z 614.286,A -85,B 0,C 180,E1 -443.484,E2 -443.484} C_VEL
LIN {X 0,Y 608.45,Z 619.865,A -85,B 0,C 180,E1 -444.365,E2 -444.365} C_VEL
LIN {X 0,Y 608.432,Z 624.949,A -85,B 0,C 180,E1 -445.362,E2 -445.362} C_VEL
LIN {X 0,Y 608.449,Z 628.896,A -85,B 0,C 180,E1 -446.357,E2 -446.357} C_VEL
LIN {X 0,Y 608.425,Z 631.809,A -85,B 0,C 180,E1 -447.352,E2 -447.352} C_VEL
LIN {X 0,Y 608.443,Z 633.201,A -85,B 0,C 180,E1 -448.014,E2 -448.014} C_VEL
LIN {X 0,Y 608.438,Z 634.783,A -85,B 0,C 180,E1 -449.338,E2 -449.338} C_VEL
LIN {X 0,Y 608.434,Z 635,A -85,B 0,C 180,E1 -450,E2 -450} C_VEL
LIN {X 0,Y 608.448,Z 634.184,A -85,B 0,C 180,E1 -451.324,E2 -451.324} C_VEL
LIN {X 0,Y 608.443,Z 633.202,A -85,B 0,C 180,E1 -451.986,E2 -451.986} C_VEL
LIN {X 0,Y 608.425,Z 631.809,A -85,B 0,C 180,E1 -452.648,E2 -452.648} C_VEL
LIN {X 0,Y 608.449,Z 628.896,A -85,B 0,C 180,E1 -453.642,E2 -453.642} C_VEL
LIN {X 0,Y 608.432,Z 624.95,A -85,B 0,C 180,E1 -454.638,E2 -454.638} C_VEL
LIN {X 0,Y 608.437,Z 618.877,A -85,B 0,C 180,E1 -455.801,E2 -455.801} C_VEL
LIN {X 0,Y 608.462,Z 612.235,A -85,B 0,C 180,E1 -456.799,E2 -456.799} C_VEL
LIN {X 0,Y 608.456,Z 603.99,A -85,B 0,C 180,E1 -457.8,E2 -457.8} C_VEL
LIN {X 0,Y 608.472,Z 595.537,A -85,B 0,C 180,E1 -458.636,E2 -458.636} C_VEL
LIN {X 0,Y 608.471,Z 585.091,A -85,B 0,C 180,E1 -459.473,E2 -459.473} C_VEL
LIN {X 0,Y 608.494,Z 574.756,A -85,B 0,C 180,E1 -460.145,E2 -460.145} C_VEL
LIN {X 0,Y 608.521,Z 563.253,A -85,B 0,C 180,E1 -460.741,E2 -460.741} C_VEL
LIN {X 0,Y 608.531,Z 550.882,A -85,B 0,C 180,E1 -461.225,E2 -461.225} C_VEL
LIN {X 0,Y 608.537,Z 537.44,A -85,B 0,C 180,E1 -461.597,E2 -461.597} C_VEL
LIN {X 0,Y 608.547,Z 525.086,A -85,B 0,C 180,E1 -461.808,E2 -461.808} C_VEL
LIN {X 0,Y 608.51,Z 421.355,A -85,B 0,C 180,E1 -463.037,E2 -463.037} C_VEL
LIN {X 0,Y 608.532,Z 395.645,A -85,B 0,C 180,E1 -465.748,E2 -465.748} C_VEL
LIN {X 0,Y 608.571,Z 368.97,A -85,B 0,C 180,E1 -468.614,E2 -468.614} C_VEL
LIN {X 0,Y 608.62,Z 344.101,A -85,B 0,C 180,E1 -471.33,E2 -471.33} C_VEL
LIN {X 0,Y 608.68,Z 318.364,A -85,B 0,C 180,E1 -474.194,E2 -474.194} C_VEL
LIN {X 0,Y 608.506,Z 305.877,A -85,B 0,C 180,E1 -475.616,E2 -475.616} C_VEL
LIN {X 0,Y 608.473,Z 305.694,A -85,B 0,C 180,E1 -478.619,E2 -478.619} C_VEL
LIN {X 0,Y 608.441,Z 305.689,A -85,B 0,C 180,E1 -481.318,E2 -481.318} C_VEL
LIN {X 0,Y 608.449,Z 305.689,A -85,B 0,C 180,E1 -483.731,E2 -483.731} C_VEL
LIN {X 0,Y 608.463,Z 305.692,A -85,B 0,C 180,E1 -486.091,E2 -486.091} C_VEL
LIN {X 0,Y 608.423,Z 305.697,A -85,B 0,C 180,E1 -488.592,E2 -488.592} C_VEL
LIN {X 0,Y 608.436,Z 305.69,A -85,B 0,C 180,E1 -491.339,E2 -491.339} C_VEL
LIN {X 0,Y 608.459,Z 305.696,A -85,B 0,C 180,E1 -494.264,E2 -494.264} C_VEL
LIN {X 0,Y 608.437,Z 305.691,A -85,B 0,C 180,E1 -496.695,E2 -496.695} C_VEL
LIN {X 0,Y 608.409,Z 305.694,A -85,B 0,C 180,E1 -498.819,E2 -498.819} C_VEL
LIN {X 0,Y 608.463,Z 305.693,A -85,B 0,C 180,E1 -501.761,E2 -501.761} C_VEL
LIN {X 0,Y 608.408,Z 305.694,A -85,B 0,C 180,E1 -504.72,E2 -504.72} C_VEL
LIN {X 0,Y 608.455,Z 305.691,A -85,B 0,C 180,E1 -507.479,E2 -507.479} C_VEL
LIN {X 0,Y 608.434,Z 305.694,A -85,B 0,C 180,E1 -510.218,E2 -510.218} C_VEL
LIN {X 0,Y 608.406,Z 305.693,A -85,B 0,C 180,E1 -512.807,E2 -512.807} C_VEL
LIN {X 0,Y 608.43,Z 305.696,A -85,B 0,C 180,E1 -515.428,E2 -515.428} C_VEL
LIN {X 0,Y 608.445,Z 305.699,A -85,B 0,C 180,E1 -517.593,E2 -517.593} C_VEL
LIN {X 0,Y 608.44,Z 305.697,A -85,B 0,C 180,E1 -519.725,E2 -519.725} C_VEL
LIN {X 0,Y 608.416,Z 305.698,A -85,B 0,C 180,E1 -521.827,E2 -521.827} C_VEL
LIN {X 0,Y 608.431,Z 305.694,A -85,B 0,C 180,E1 -523.905,E2 -523.905} C_VEL
LIN {X 0,Y 608.412,Z 305.693,A -85,B 0,C 180,E1 -526.642,E2 -526.642} C_VEL
LIN {X 0,Y 608.458,Z 305.694,A -85,B 0,C 180,E1 -529.173,E2 -529.173} C_VEL
LIN {X 0,Y 608.478,Z 400.742,A -85,B 0,C 180,E1 -530.317,E2 -530.317} C_VEL
LIN {X 0,Y 608.47,Z 414.018,A -85,B 0,C 180,E1 -530.61,E2 -530.61} C_VEL
LIN {X 0,Y 608.508,Z 426.7,A -85,B 0,C 180,E1 -531.03,E2 -531.03} C_VEL
LIN {X 0,Y 608.522,Z 437.992,A -85,B 0,C 180,E1 -531.532,E2 -531.532} C_VEL
LIN {X 0,Y 608.477,Z 449.641,A -85,B 0,C 180,E1 -532.2,E2 -532.2} C_VEL
LIN {X 0,Y 608.486,Z 460.083,A -85,B 0,C 180,E1 -532.951,E2 -532.951} C_VEL
LIN {X 0,Y 608.461,Z 468.648,A -85,B 0,C 180,E1 -533.7,E2 -533.7} C_VEL
LIN {X 0,Y 608.462,Z 476.545,A -85,B 0,C 180,E1 -534.532,E2 -534.532} C_VEL
LIN {X 0,Y 608.448,Z 484.276,A -85,B 0,C 180,E1 -535.528,E2 -535.528} C_VEL
LIN {X 0,Y 608.434,Z 491.383,A -85,B 0,C 180,E1 -536.689,E2 -536.689} C_VEL
LIN {X 0,Y 608.457,Z 496.127,A -85,B 0,C 180,E1 -537.683,E2 -537.683} C_VEL
LIN {X 0,Y 608.45,Z 499.769,A -85,B 0,C 180,E1 -538.676,E2 -538.676} C_VEL
LIN {X 0,Y 608.438,Z 501.654,A -85,B 0,C 180,E1 -539.338,E2 -539.338} C_VEL
LIN {X 0,Y 608.434,Z 503.103,A -85,B 0,C 180,E1 -540,E2 -540} C_VEL
LIN {X 0,Y 608.447,Z 504.742,A -85,B 0,C 180,E1 -541.323,E2 -541.323} C_VEL
LIN {X 0,Y 608.442,Z 504.992,A -85,B 0,C 180,E1 -541.986,E2 -541.986} C_VEL
LIN {X 0,Y 608.423,Z 504.825,A -85,B 0,C 180,E1 -542.648,E2 -542.648} C_VEL
LIN {X 0,Y 608.433,Z 503.296,A -85,B 0,C 180,E1 -543.974,E2 -543.974} C_VEL
LIN {X 0,Y 608.431,Z 501.941,A -85,B 0,C 180,E1 -544.638,E2 -544.638} C_VEL
LIN {X 0,Y 608.427,Z 499.066,A -85,B 0,C 180,E1 -545.634,E2 -545.634} C_VEL
LIN {X 0,Y 608.44,Z 495.163,A -85,B 0,C 180,E1 -546.633,E2 -546.633} C_VEL
LIN {X 0,Y 608.45,Z 490.118,A -85,B 0,C 180,E1 -547.633,E2 -547.633} C_VEL
LIN {X 0,Y 608.453,Z 483.774,A -85,B 0,C 180,E1 -548.636,E2 -548.636} C_VEL
LIN {X 0,Y 608.468,Z 480.16,A -85,B 0,C 180,E1 -549.119,E2 -549.119} C_VEL
LIN {X 0,Y 607.854,Z 476.644,A -85,B 0,C 180,E1 -549.562,E2 -549.562} C_VEL
LIN {X 0,Y 605.022,Z 470.606,A -85,B 0,C 180,E1 -550.256,E2 -550.256} C_VEL
LIN {X 0,Y 602.139,Z 464.022,A -85,B 0,C 180,E1 -550.908,E2 -550.908} C_VEL
LIN {X 0,Y 601.449,Z 459.644,A -85,B 0,C 180,E1 -551.282,E2 -551.282} C_VEL
LIN {X 0,Y 601.463,Z 448.882,A -85,B 0,C 180,E1 -552.056,E2 -552.056} C_VEL
LIN {X 0,Y 601.502,Z 438.511,A -85,B 0,C 180,E1 -552.654,E2 -552.654} C_VEL
LIN {X 0,Y 601.542,Z 426.128,A -85,B 0,C 180,E1 -553.212,E2 -553.212} C_VEL
LIN {X 0,Y 601.579,Z 412.883,A -85,B 0,C 180,E1 -553.645,E2 -553.645} C_VEL
LIN {X 0,Y 601.61,Z 400.663,A -85,B 0,C 180,E1 -553.911,E2 -553.911} C_VEL
LIN {X 0,Y 601.563,Z 307.201,A -85,B 0,C 180,E1 -555.045,E2 -555.045} C_VEL
LIN {X 0,Y 601.454,Z 306.565,A -85,B 0,C 180,E1 -555.069,E2 -555.069} C_VEL
LIN {X 0,Y 601.391,Z 306.567,A -85,B 0,C 180,E1 -557.688,E2 -557.688} C_VEL
LIN {X 0,Y 601.425,Z 306.571,A -85,B 0,C 180,E1 -560.522,E2 -560.522} C_VEL
LIN {X 0,Y 601.394,Z 306.567,A -85,B 0,C 180,E1 -563.411,E2 -563.411} C_VEL
LIN {X 0,Y 601.401,Z 306.566,A -85,B 0,C 180,E1 -565.864,E2 -565.864} C_VEL
LIN {X 0,Y 601.397,Z 306.567,A -85,B 0,C 180,E1 -567.868,E2 -567.868} C_VEL
LIN {X 0,Y 601.406,Z 306.569,A -85,B 0,C 180,E1 -570.165,E2 -570.165} C_VEL
LIN {X 0,Y 601.421,Z 306.571,A -85,B 0,C 180,E1 -572.715,E2 -572.715} C_VEL
LIN {X 0,Y 601.396,Z 306.569,A -85,B 0,C 180,E1 -575.112,E2 -575.112} C_VEL
LIN {X 0,Y 601.434,Z 306.562,A -85,B 0,C 180,E1 -577.419,E2 -577.419} C_VEL
LIN {X 0,Y 601.399,Z 306.569,A -85,B 0,C 180,E1 -579.996,E2 -579.996} C_VEL
LIN {X 0,Y 601.413,Z 306.572,A -85,B 0,C 180,E1 -582.67,E2 -582.67} C_VEL
LIN {X 0,Y 601.397,Z 306.566,A -85,B 0,C 180,E1 -585.479,E2 -585.479} C_VEL
LIN {X 0,Y 601.421,Z 306.574,A -85,B 0,C 180,E1 -588.407,E2 -588.407} C_VEL
LIN {X 0,Y 601.434,Z 306.565,A -85,B 0,C 180,E1 -590.875,E2 -590.875} C_VEL
LIN {X 0,Y 601.401,Z 306.566,A -85,B 0,C 180,E1 -593.417,E2 -593.417} C_VEL
LIN {X 0,Y 601.431,Z 306.568,A -85,B 0,C 180,E1 -596.064,E2 -596.064} C_VEL
LIN {X 0,Y 601.429,Z 306.563,A -85,B 0,C 180,E1 -599.058,E2 -599.058} C_VEL
LIN {X 0,Y 601.426,Z 306.563,A -85,B 0,C 180,E1 -601.373,E2 -601.373} C_VEL
LIN {X 0,Y 601.401,Z 306.567,A -85,B 0,C 180,E1 -603.636,E2 -603.636} C_VEL
LIN {X 0,Y 601.419,Z 306.568,A -85,B 0,C 180,E1 -606.59,E2 -606.59} C_VEL
LIN {X 0,Y 601.425,Z 306.563,A -85,B 0,C 180,E1 -609.478,E2 -609.478} C_VEL
LIN {X 0,Y 601.396,Z 306.575,A -85,B 0,C 180,E1 -612.312,E2 -612.312} C_VEL
LIN {X 0,Y 601.412,Z 306.571,A -85,B 0,C 180,E1 -614.409,E2 -614.409} C_VEL
LIN {X 0,Y 601.414,Z 306.564,A -85,B 0,C 180,E1 -617.172,E2 -617.172} C_VEL
LIN {X 0,Y 601.436,Z 306.568,A -85,B 0,C 180,E1 -619.905,E2 -619.905} C_VEL
LIN {X 0,Y 601.439,Z 306.563,A -85,B 0,C 180,E1 -622.615,E2 -622.615} C_VEL
LIN {X 0,Y 601.415,Z 306.565,A -85,B 0,C 180,E1 -625.308,E2 -625.308} C_VEL
LIN {X 0,Y 601.436,Z 306.572,A -85,B 0,C 180,E1 -627.991,E2 -627.991} C_VEL
LIN {X 0,Y 601.446,Z 306.561,A -85,B 0,C 180,E1 -630.67,E2 -630.67} C_VEL
LIN {X 0,Y 601.426,Z 306.564,A -85,B 0,C 180,E1 -633.35,E2 -633.35} C_VEL
LIN {X 0,Y 601.415,Z 306.573,A -85,B 0,C 180,E1 -636.037,E2 -636.037} C_VEL
LIN {X 0,Y 601.41,Z 306.565,A -85,B 0,C 180,E1 -638.738,E2 -638.738} C_VEL
LIN {X 0,Y 601.433,Z 306.565,A -85,B 0,C 180,E1 -641.458,E2 -641.458} C_VEL
LIN {X 0,Y 601.418,Z 306.569,A -85,B 0,C 180,E1 -644.206,E2 -644.206} C_VEL
LIN {X 0,Y 601.429,Z 306.563,A -85,B 0,C 180,E1 -646.986,E2 -646.986} C_VEL
LIN {X 0,Y 601.401,Z 306.576,A -85,B 0,C 180,E1 -649.81,E2 -649.81} C_VEL
LIN {X 0,Y 601.411,Z 306.565,A -85,B 0,C 180,E1 -652.683,E2 -652.683} C_VEL
LIN {X 0,Y 601.401,Z 306.566,A -85,B 0,C 180,E1 -654.879,E2 -654.879} C_VEL
LIN {X 0,Y 601.416,Z 306.573,A -85,B 0,C 180,E1 -657.868,E2 -657.868} C_VEL
LIN {X 0,Y 601.427,Z 306.566,A -85,B 0,C 180,E1 -660.164,E2 -660.164} C_VEL
LIN {X 0,Y 601.415,Z 306.564,A -85,B 0,C 180,E1 -662.715,E2 -662.715} C_VEL
LIN {X 0,Y 601.421,Z 306.565,A -85,B 0,C 180,E1 -665.116,E2 -665.116} C_VEL
LIN {X 0,Y 601.433,Z 306.568,A -85,B 0,C 180,E1 -667.42,E2 -667.42} C_VEL
LIN {X 0,Y 601.411,Z 306.569,A -85,B 0,C 180,E1 -669.996,E2 -669.996} C_VEL
LIN {X 0,Y 601.407,Z 306.565,A -85,B 0,C 180,E1 -672.671,E2 -672.671} C_VEL
LIN {X 0,Y 601.427,Z 306.572,A -85,B 0,C 180,E1 -675.483,E2 -675.483} C_VEL
LIN {X 0,Y 601.421,Z 306.564,A -85,B 0,C 180,E1 -678.408,E2 -678.408} C_VEL
LIN {X 0,Y 601.412,Z 306.566,A -85,B 0,C 180,E1 -680.874,E2 -680.874} C_VEL
LIN {X 0,Y 601.403,Z 306.575,A -85,B 0,C 180,E1 -683.417,E2 -683.417} C_VEL
LIN {X 0,Y 601.418,Z 306.566,A -85,B 0,C 180,E1 -686.067,E2 -686.067} C_VEL
LIN {X 0,Y 601.421,Z 306.563,A -85,B 0,C 180,E1 -688.546,E2 -688.546} C_VEL
LIN {X 0,Y 601.433,Z 306.572,A -85,B 0,C 180,E1 -691.374,E2 -691.374} C_VEL
LIN {X 0,Y 601.398,Z 306.573,A -85,B 0,C 180,E1 -693.636,E2 -693.636} C_VEL
LIN {X 0,Y 601.442,Z 306.564,A -85,B 0,C 180,E1 -695.859,E2 -695.859} C_VEL
LIN {X 0,Y 601.409,Z 306.567,A -85,B 0,C 180,E1 -698.761,E2 -698.761} C_VEL
LIN {X 0,Y 601.425,Z 306.568,A -85,B 0,C 180,E1 -699.03,E2 -699.03} C_VEL
LIN {X 0,Y 601.644,Z 310.306,A -85,B 0,C 180,E1 -699.084,E2 -699.084} C_VEL
LIN {X 0,Y 601.584,Z 401.657,A -85,B 0,C 180,E1 -700.197,E2 -700.197} C_VEL
LIN {X 0,Y 601.578,Z 415.117,A -85,B 0,C 180,E1 -700.508,E2 -700.508} C_VEL
LIN {X 0,Y 601.562,Z 428.057,A -85,B 0,C 180,E1 -700.954,E2 -700.954} C_VEL
LIN {X 0,Y 601.511,Z 439.664,A -85,B 0,C 180,E1 -701.498,E2 -701.498} C_VEL
LIN {X 0,Y 601.458,Z 450.456,A -85,B 0,C 180,E1 -702.138,E2 -702.138} C_VEL
LIN {X 0,Y 601.458,Z 461.135,A -85,B 0,C 180,E1 -702.928,E2 -702.928} C_VEL
LIN {X 0,Y 601.409,Z 469.802,A -85,B 0,C 180,E1 -703.713,E2 -703.713} C_VEL
LIN {X 0,Y 601.381,Z 479.106,A -85,B 0,C 180,E1 -704.755,E2 -704.755} C_VEL
LIN {X 0,Y 601.384,Z 486.545,A -85,B 0,C 180,E1 -705.794,E2 -705.794} C_VEL
LIN {X 0,Y 601.35,Z 492.451,A -85,B 0,C 180,E1 -706.827,E2 -706.827} C_VEL
LIN {X 0,Y 601.367,Z 497.061,A -85,B 0,C 180,E1 -707.857,E2 -707.857} C_VEL
LIN {X 0,Y 601.336,Z 500.94,A -85,B 0,C 180,E1 -709.034,E2 -709.034} C_VEL
LIN {X 0,Y 601.328,Z 502.969,A -85,B 0,C 180,E1 -709.904,E2 -709.904} C_VEL
LIN {X 0,Y 601.336,Z 504.041,A -85,B 0,C 180,E1 -710.583,E2 -710.583} C_VEL
LIN {X 0,Y 601.332,Z 504.981,A -85,B 0,C 180,E1 -711.938,E2 -711.938} C_VEL
LIN {X 0,Y 601.322,Z 504.847,A -85,B 0,C 180,E1 -712.614,E2 -712.614} C_VEL
LIN {X 0,Y 601.349,Z 504.145,A -85,B 0,C 180,E1 -713.417,E2 -713.417} C_VEL
LIN {X 0,Y 601.349,Z 502.006,A -85,B 0,C 180,E1 -714.636,E2 -714.636} C_VEL
LIN {X 0,Y 601.355,Z 499.166,A -85,B 0,C 180,E1 -715.644,E2 -715.644} C_VEL
LIN {X 0,Y 601.349,Z 495.31,A -85,B 0,C 180,E1 -716.65,E2 -716.65} C_VEL
LIN {X 0,Y 601.366,Z 490.346,A -85,B 0,C 180,E1 -717.656,E2 -717.656} C_VEL
LIN {X 0,Y 601.385,Z 484.127,A -85,B 0,C 180,E1 -718.661,E2 -718.661} C_VEL
LIN {X 0,Y 601.414,Z 476.382,A -85,B 0,C 180,E1 -719.666,E2 -719.666} C_VEL
LIN {X 0,Y 601.432,Z 466.742,A -85,B 0,C 180,E1 -720.67,E2 -720.67} C_VEL
LIN {X 0,Y 601.469,Z 456.772,A -85,B 0,C 180,E1 -721.507,E2 -721.507} C_VEL
LIN {X 0,Y 601.475,Z 445.575,A -85,B 0,C 180,E1 -722.26,E2 -722.26} C_VEL
LIN {X 0,Y 601.524,Z 434.621,A -85,B 0,C 180,E1 -722.847,E2 -722.847} C_VEL
LIN {X 0,Y 601.536,Z 422.428,A -85,B 0,C 180,E1 -723.349,E2 -723.349} C_VEL
LIN {X 0,Y 601.529,Z 409.666,A -85,B 0,C 180,E1 -723.727,E2 -723.727} C_VEL
LIN {X 0,Y 601.559,Z 396.086,A -85,B 0,C 180,E1 -723.978,E2 -723.978} C_VEL
LIN {X 0,Y 601.583,Z 307.445,A -85,B 0,C 180,E1 -725.041,E2 -725.041} C_VEL
LIN {X 0,Y 601.416,Z 306.569,A -85,B 0,C 180,E1 -725.07,E2 -725.07} C_VEL
LIN {X 0,Y 601.368,Z 306.571,A -85,B 0,C 180,E1 -727.386,E2 -727.386} C_VEL
LIN {X 0,Y 601.369,Z 306.571,A -85,B 0,C 180,E1 -729.417,E2 -729.417} C_VEL
LIN {X 0,Y 601.392,Z 306.571,A -85,B 0,C 180,E1 -732.143,E2 -732.143} C_VEL
LIN {X 0,Y 601.391,Z 306.571,A -85,B 0,C 180,E1 -734.898,E2 -734.898} C_VEL
LIN {X 0,Y 601.372,Z 306.572,A -85,B 0,C 180,E1 -736.988,E2 -736.988} C_VEL
LIN {X 0,Y 601.367,Z 306.572,A -85,B 0,C 180,E1 -739.811,E2 -739.811} C_VEL
LIN {X 0,Y 601.41,Z 306.569,A -85,B 0,C 180,E1 -742.683,E2 -742.683} C_VEL
LIN {X 0,Y 601.368,Z 306.572,A -85,B 0,C 180,E1 -744.88,E2 -744.88} C_VEL
LIN {X 0,Y 601.361,Z 306.571,A -85,B 0,C 180,E1 -747.351,E2 -747.351} C_VEL
LIN {X 0,Y 601.407,Z 306.576,A -85,B 0,C 180,E1 -750.166,E2 -750.166} C_VEL
LIN {X 0,Y 601.409,Z 306.567,A -85,B 0,C 180,E1 -752.713,E2 -752.713} C_VEL
LIN {X 0,Y 601.363,Z 306.571,A -85,B 0,C 180,E1 -755.107,E2 -755.107} C_VEL
LIN {X 0,Y 601.393,Z 306.569,A -85,B 0,C 180,E1 -757.422,E2 -757.422} C_VEL
LIN {X 0,Y 601.4,Z 306.576,A -85,B 0,C 180,E1 -759.996,E2 -759.996} C_VEL
LIN {X 0,Y 601.381,Z 306.569,A -85,B 0,C 180,E1 -762.673,E2 -762.673} C_VEL
LIN {X 0,Y 601.403,Z 306.57,A -85,B 0,C 180,E1 -765.479,E2 -765.479} C_VEL
LIN {X 0,Y 601.415,Z 306.566,A -85,B 0,C 180,E1 -768.408,E2 -768.408} C_VEL
LIN {X 0,Y 601.392,Z 306.567,A -85,B 0,C 180,E1 -770.872,E2 -770.872} C_VEL
LIN {X 0,Y 601.398,Z 306.575,A -85,B 0,C 180,E1 -773.74,E2 -773.74} C_VEL
LIN {X 0,Y 601.414,Z 306.565,A -85,B 0,C 180,E1 -776.685,E2 -776.685} C_VEL
LIN {X 0,Y 601.407,Z 306.568,A -85,B 0,C 180,E1 -779.057,E2 -779.057} C_VEL
LIN {X 0,Y 601.43,Z 306.571,A -85,B 0,C 180,E1 -781.373,E2 -781.373} C_VEL
LIN {X 0,Y 601.415,Z 306.595,A -85,B 0,C 180,E1 -784.143,E2 -784.143} C_VEL
LIN {X 0,Y 601.897,Z 310.274,A -85,B 0,C 180,E1 -784.589,E2 -784.589} C_VEL
LIN {X 0,Y 601.79,Z 334.435,A -85,B 0,C 180,E1 -787.332,E2 -787.332} C_VEL
LIN {X 0,Y 601.716,Z 358.596,A -85,B 0,C 180,E1 -790.023,E2 -790.023} C_VEL
LIN {X 0,Y 601.594,Z 385.978,A -85,B 0,C 180,E1 -793.019,E2 -793.019} C_VEL
LIN {X 0,Y 601.52,Z 413.694,A -85,B 0,C 180,E1 -796.005,E2 -796.005} C_VEL
LIN {X 0,Y 601.514,Z 421.336,A -85,B 0,C 180,E1 -796.809,E2 -796.809} C_VEL
LIN {X 0,Y 601.605,Z 530.936,A -85,B 0,C 180,E1 -798.139,E2 -798.139} C_VEL
LIN {X 0,Y 601.574,Z 544.21,A -85,B 0,C 180,E1 -798.438,E2 -798.438} C_VEL
LIN {X 0,Y 601.544,Z 555.964,A -85,B 0,C 180,E1 -798.828,E2 -798.828} C_VEL
LIN {X 0,Y 601.516,Z 566.919,A -85,B 0,C 180,E1 -799.311,E2 -799.311} C_VEL
LIN {X 0,Y 601.479,Z 577.577,A -85,B 0,C 180,E1 -799.906,E2 -799.906} C_VEL
LIN {X 0,Y 601.446,Z 588.473,A -85,B 0,C 180,E1 -800.669,E2 -800.669} C_VEL
LIN {X 0,Y 601.429,Z 599.11,A -85,B 0,C 180,E1 -801.601,E2 -801.601} C_VEL
LIN {X 0,Y 601.418,Z 606.959,A -85,B 0,C 180,E1 -802.446,E2 -802.446} C_VEL
LIN {X 0,Y 601.37,Z 614.224,A -85,B 0,C 180,E1 -803.398,E2 -803.398} C_VEL
LIN {X 0,Y 601.372,Z 619.865,A -85,B 0,C 180,E1 -804.299,E2 -804.299} C_VEL
LIN {X 0,Y 601.337,Z 624.949,A -85,B 0,C 180,E1 -805.307,E2 -805.307} C_VEL
LIN {X 0,Y 601.367,Z 628.896,A -85,B 0,C 180,E1 -806.315,E2 -806.315} C_VEL
LIN {X 0,Y 601.325,Z 631.809,A -85,B 0,C 180,E1 -807.32,E2 -807.32} C_VEL
LIN {X 0,Y 601.341,Z 633.201,A -85,B 0,C 180,E1 -807.991,E2 -807.991} C_VEL
LIN {X 0,Y 601.339,Z 634.784,A -85,B 0,C 180,E1 -809.33,E2 -809.33} C_VEL
LIN {X 0,Y 601.335,Z 635,A -85,B 0,C 180,E1 -810,E2 -810} C_VEL
LIN {X 0,Y 601.348,Z 634.184,A -85,B 0,C 180,E1 -811.339,E2 -811.339} C_VEL
LIN {X 0,Y 601.341,Z 633.202,A -85,B 0,C 180,E1 -812.009,E2 -812.009} C_VEL
LIN {X 0,Y 601.325,Z 631.81,A -85,B 0,C 180,E1 -812.679,E2 -812.679} C_VEL
LIN {X 0,Y 601.367,Z 628.896,A -85,B 0,C 180,E1 -813.685,E2 -813.685} C_VEL
LIN {X 0,Y 601.337,Z 624.95,A -85,B 0,C 180,E1 -814.693,E2 -814.693} C_VEL
LIN {X 0,Y 601.372,Z 618.877,A -85,B 0,C 180,E1 -815.869,E2 -815.869} C_VEL
LIN {X 0,Y 601.382,Z 612.236,A -85,B 0,C 180,E1 -816.88,E2 -816.88} C_VEL
LIN {X 0,Y 601.4,Z 603.99,A -85,B 0,C 180,E1 -817.892,E2 -817.892} C_VEL
LIN {X 0,Y 601.436,Z 595.537,A -85,B 0,C 180,E1 -818.738,E2 -818.738} C_VEL
LIN {X 0,Y 601.442,Z 585.093,A -85,B 0,C 180,E1 -819.585,E2 -819.585} C_VEL
LIN {X 0,Y 601.472,Z 574.758,A -85,B 0,C 180,E1 -820.264,E2 -820.264} C_VEL
LIN {X 0,Y 601.536,Z 563.905,A -85,B 0,C 180,E1 -820.836,E2 -820.836} C_VEL
LIN {X 0,Y 601.557,Z 551.379,A -85,B 0,C 180,E1 -821.34,E2 -821.34} C_VEL
LIN {X 0,Y 601.569,Z 538.353,A -85,B 0,C 180,E1 -821.712,E2 -821.712} C_VEL
LIN {X 0,Y 601.614,Z 525.086,A -85,B 0,C 180,E1 -821.946,E2 -821.946} C_VEL
LIN {X 0,Y 601.514,Z 421.355,A -85,B 0,C 180,E1 -823.191,E2 -823.191} C_VEL
LIN {X 0,Y 601.553,Z 395.645,A -85,B 0,C 180,E1 -825.935,E2 -825.935} C_VEL
LIN {X 0,Y 601.633,Z 373.095,A -85,B 0,C 180,E1 -828.385,E2 -828.385} C_VEL
LIN {X 0,Y 601.725,Z 349.499,A -85,B 0,C 180,E1 -830.985,E2 -830.985} C_VEL
LIN {X 0,Y 601.833,Z 324.772,A -85,B 0,C 180,E1 -833.758,E2 -833.758} C_VEL
LIN {X 0,Y 601.834,Z 308.665,A -85,B 0,C 180,E1 -835.599,E2 -835.599} C_VEL
LIN {X 0,Y 601.424,Z 306.569,A -85,B 0,C 180,E1 -835.869,E2 -835.869} C_VEL
LIN {X 0,Y 601.428,Z 306.569,A -85,B 0,C 180,E1 -838.787,E2 -838.787} C_VEL
LIN {X 0,Y 601.418,Z 306.564,A -85,B 0,C 180,E1 -841.454,E2 -841.454} C_VEL
LIN {X 0,Y 601.418,Z 306.57,A -85,B 0,C 180,E1 -844.119,E2 -844.119} C_VEL
LIN {X 0,Y 601.392,Z 306.573,A -85,B 0,C 180,E1 -846.584,E2 -846.584} C_VEL
LIN {X 0,Y 601.391,Z 306.568,A -85,B 0,C 180,E1 -849.128,E2 -849.128} C_VEL
LIN {X 0,Y 601.423,Z 306.567,A -85,B 0,C 180,E1 -851.765,E2 -851.765} C_VEL
LIN {X 0,Y 601.401,Z 306.57,A -85,B 0,C 180,E1 -854.532,E2 -854.532} C_VEL
LIN {X 0,Y 601.387,Z 306.569,A -85,B 0,C 180,E1 -857.412,E2 -857.412} C_VEL
LIN {X 0,Y 601.398,Z 306.577,A -85,B 0,C 180,E1 -860.004,E2 -860.004} C_VEL
LIN {X 0,Y 601.392,Z 306.568,A -85,B 0,C 180,E1 -862.624,E2 -862.624} C_VEL
LIN {X 0,Y 601.373,Z 306.57,A -85,B 0,C 180,E1 -865.065,E2 -865.065} C_VEL
LIN {X 0,Y 601.424,Z 306.567,A -85,B 0,C 180,E1 -867.484,E2 -867.484} C_VEL
LIN {X 0,Y 601.405,Z 306.576,A -85,B 0,C 180,E1 -869.856,E2 -869.856} C_VEL
LIN {X 0,Y 601.361,Z 306.571,A -85,B 0,C 180,E1 -872.648,E2 -872.648} C_VEL
LIN {X 0,Y 601.366,Z 306.573,A -85,B 0,C 180,E1 -875.12,E2 -875.12} C_VEL
LIN {X 0,Y 601.418,Z 306.57,A -85,B 0,C 180,E1 -877.395,E2 -877.395} C_VEL
LIN {X 0,Y 601.368,Z 306.572,A -85,B 0,C 180,E1 -880.189,E2 -880.189} C_VEL
LIN {X 0,Y 601.373,Z 306.572,A -85,B 0,C 180,E1 -883.012,E2 -883.012} C_VEL
LIN {X 0,Y 601.376,Z 306.573,A -85,B 0,C 180,E1 -885.927,E2 -885.927} C_VEL
LIN {X 0,Y 601.373,Z 306.57,A -85,B 0,C 180,E1 -888.54,E2 -888.54} C_VEL
LIN {X 0,Y 601.396,Z 306.572,A -85,B 0,C 180,E1 -889.026,E2 -889.026} C_VEL
LIN {X 0,Y 601.652,Z 310.35,A -85,B 0,C 180,E1 -889.085,E2 -889.085} C_VEL
LIN {X 0,Y 601.534,Z 400.919,A -85,B 0,C 180,E1 -890.182,E2 -890.182} C_VEL
LIN {X 0,Y 601.522,Z 414.137,A -85,B 0,C 180,E1 -890.479,E2 -890.479} C_VEL
LIN {X 0,Y 601.536,Z 427.346,A -85,B 0,C 180,E1 -890.925,E2 -890.925} C_VEL
LIN {X 0,Y 601.537,Z 438.452,A -85,B 0,C 180,E1 -891.433,E2 -891.433} C_VEL
LIN {X 0,Y 601.448,Z 450.003,A -85,B 0,C 180,E1 -892.108,E2 -892.108} C_VEL
LIN {X 0,Y 601.463,Z 460.385,A -85,B 0,C 180,E1 -892.868,E2 -892.868} C_VEL
LIN {X 0,Y 601.416,Z 470.407,A -85,B 0,C 180,E1 -893.775,E2 -893.775} C_VEL
LIN {X 0,Y 601.384,Z 479.492,A -85,B 0,C 180,E1 -894.803,E2 -894.803} C_VEL
LIN {X 0,Y 601.365,Z 486.655,A -85,B 0,C 180,E1 -895.811,E2 -895.811} C_VEL
LIN {X 0,Y 601.352,Z 491.51,A -85,B 0,C 180,E1 -896.65,E2 -896.65} C_VEL
LIN {X 0,Y 601.364,Z 496.223,A -85,B 0,C 180,E1 -897.655,E2 -897.655} C_VEL
LIN {X 0,Y 601.351,Z 499.84,A -85,B 0,C 180,E1 -898.66,E2 -898.66} C_VEL
LIN {X 0,Y 601.339,Z 501.718,A -85,B 0,C 180,E1 -899.33,E2 -899.33} C_VEL
LIN {X 0,Y 601.335,Z 503.144,A -85,B 0,C 180,E1 -900,E2 -900} C_VEL
LIN {X 0,Y 601.347,Z 504.759,A -85,B 0,C 180,E1 -901.339,E2 -901.339} C_VEL
LIN {X 0,Y 601.341,Z 504.997,A -85,B 0,C 180,E1 -902.009,E2 -902.009} C_VEL
LIN {X 0,Y 601.338,Z 504.223,A -85,B 0,C 180,E1 -903.35,E2 -903.35} C_VEL
LIN {X 0,Y 601.342,Z 503.258,A -85,B 0,C 180,E1 -904.021,E2 -904.021} C_VEL
LIN {X 0,Y 601.33,Z 501.877,A -85,B 0,C 180,E1 -904.692,E2 -904.692} C_VEL
LIN {X 0,Y 601.356,Z 498.982,A -85,B 0,C 180,E1 -905.701,E2 -905.701} C_VEL
LIN {X 0,Y 601.356,Z 495.053,A -85,B 0,C 180,E1 -906.711,E2 -906.711} C_VEL
LIN {X 0,Y 601.385,Z 489.983,A -85,B 0,C 180,E1 -907.723,E2 -907.723} C_VEL
LIN {X 0,Y 601.386,Z 483.602,A -85,B 0,C 180,E1 -908.738,E2 -908.738} C_VEL
LIN {X 0,Y 601.397,Z 475.591,A -85,B 0,C 180,E1 -909.755,E2 -909.755} C_VEL
LIN {X 0,Y 601.417,Z 467.42,A -85,B 0,C 180,E1 -910.605,E2 -910.605} C_VEL
LIN {X 0,Y 601.449,Z 459.644,A -85,B 0,C 180,E1 -911.282,E2 -911.282} C_VEL
LIN {X 0,Y 600.775,Z 455.147,A -85,B 0,C 180,E1 -911.639,E2 -911.639} C_VEL
LIN {X 0,Y 597.958,Z 447.629,A -85,B 0,C 180,E1 -912.196,E2 -912.196} C_VEL
LIN {X 0,Y 595.176,Z 439.73,A -85,B 0,C 180,E1 -912.703,E2 -912.703} C_VEL
LIN {X 0,Y 594.555,Z 434.567,A -85,B 0,C 180,E1 -912.978,E2 -912.978} C_VEL
LIN {X 0,Y 594.584,Z 423.186,A -85,B 0,C 180,E1 -913.456,E2 -913.456} C_VEL
LIN {X 0,Y 594.639,Z 410.593,A -85,B 0,C 180,E1 -913.84,E2 -913.84} C_VEL
LIN {X 0,Y 594.676,Z 397.417,A -85,B 0,C 180,E1 -914.099,E2 -914.099} C_VEL
LIN {X 0,Y 594.697,Z 308.742,A -85,B 0,C 180,E1 -915.179,E2 -915.179} C_VEL
LIN {X 0,Y 594.393,Z 307.443,A -85,B 0,C 180,E1 -915.209,E2 -915.209} C_VEL
LIN {X 0,Y 594.343,Z 307.446,A -85,B 0,C 180,E1 -917.905,E2 -917.905} C_VEL
LIN {X 0,Y 594.404,Z 307.447,A -85,B 0,C 180,E1 -920.775,E2 -920.775} C_VEL
LIN {X 0,Y 594.37,Z 307.442,A -85,B 0,C 180,E1 -923.704,E2 -923.704} C_VEL
LIN {X 0,Y 594.382,Z 307.45,A -85,B 0,C 180,E1 -926.699,E2 -926.699} C_VEL
LIN {X 0,Y 594.381,Z 307.444,A -85,B 0,C 180,E1 -928.998,E2 -928.998} C_VEL
LIN {X 0,Y 594.376,Z 307.441,A -85,B 0,C 180,E1 -931.642,E2 -931.642} C_VEL
LIN {X 0,Y 594.379,Z 307.451,A -85,B 0,C 180,E1 -934.58,E2 -934.58} C_VEL
LIN {X 0,Y 594.387,Z 307.44,A -85,B 0,C 180,E1 -937.608,E2 -937.608} C_VEL
LIN {X 0,Y 594.366,Z 307.452,A -85,B 0,C 180,E1 -940.567,E2 -940.567} C_VEL
LIN {X 0,Y 594.367,Z 307.442,A -85,B 0,C 180,E1 -943.299,E2 -943.299} C_VEL
LIN {X 0,Y 594.358,Z 307.449,A -85,B 0,C 180,E1 -946.161,E2 -946.161} C_VEL
LIN {X 0,Y 594.379,Z 307.449,A -85,B 0,C 180,E1 -948.536,E2 -948.536} C_VEL
LIN {X 0,Y 594.384,Z 307.44,A -85,B 0,C 180,E1 -951.295,E2 -951.295} C_VEL
LIN {X 0,Y 594.35,Z 307.446,A -85,B 0,C 180,E1 -953.755,E2 -953.755} C_VEL
LIN {X 0,Y 594.378,Z 307.45,A -85,B 0,C 180,E1 -956.239,E2 -956.239} C_VEL
LIN {X 0,Y 594.389,Z 307.444,A -85,B 0,C 180,E1 -958.651,E2 -958.651} C_VEL
LIN {X 0,Y 594.381,Z 307.441,A -85,B 0,C 180,E1 -961.042,E2 -961.042} C_VEL
LIN {X 0,Y 594.389,Z 307.445,A -85,B 0,C 180,E1 -963.976,E2 -963.976} C_VEL
LIN {X 0,Y 594.385,Z 307.45,A -85,B 0,C 180,E1 -966.296,E2 -966.296} C_VEL
LIN {X 0,Y 594.4,Z 307.438,A -85,B 0,C 180,E1 -969.224,E2 -969.224} C_VEL
LIN {X 0,Y 594.377,Z 307.45,A -85,B 0,C 180,E1 -972.096,E2 -972.096} C_VEL
LIN {X 0,Y 594.365,Z 307.452,A -85,B 0,C 180,E1 -974.219,E2 -974.219} C_VEL
LIN {X 0,Y 594.382,Z 307.448,A -85,B 0,C 180,E1 -976.321,E2 -976.321} C_VEL
LIN {X 0,Y 594.373,Z 307.441,A -85,B 0,C 180,E1 -979.095,E2 -979.095} C_VEL
LIN {X 0,Y 594.411,Z 307.443,A -85,B 0,C 180,E1 -981.843,E2 -981.843} C_VEL
LIN {X 0,Y 594.392,Z 307.442,A -85,B 0,C 180,E1 -984.572,E2 -984.572} C_VEL
LIN {X 0,Y 594.402,Z 307.438,A -85,B 0,C 180,E1 -987.289,E2 -987.289} C_VEL
LIN {X 0,Y 594.414,Z 307.447,A -85,B 0,C 180,E1 -990,E2 -990} C_VEL
LIN {X 0,Y 594.402,Z 307.439,A -85,B 0,C 180,E1 -992.711,E2 -992.711} C_VEL
LIN {X 0,Y 594.391,Z 307.441,A -85,B 0,C 180,E1 -995.428,E2 -995.428} C_VEL
LIN {X 0,Y 594.412,Z 307.443,A -85,B 0,C 180,E1 -998.157,E2 -998.157} C_VEL
LIN {X 0,Y 594.388,Z 307.44,A -85,B 0,C 180,E1 -1001.075,E2 -1001.075} C_VEL
LIN {X 0,Y 594.382,Z 307.447,A -85,B 0,C 180,E1 -1003.679,E2 -1003.679} C_VEL
LIN {X 0,Y 594.389,Z 307.44,A -85,B 0,C 180,E1 -1006.719,E2 -1006.719} C_VEL
LIN {X 0,Y 594.365,Z 307.445,A -85,B 0,C 180,E1 -1009.335,E2 -1009.335} C_VEL
LIN {X 0,Y 594.362,Z 307.448,A -85,B 0,C 180,E1 -1011.504,E2 -1011.504} C_VEL
LIN {X 0,Y 594.387,Z 307.441,A -85,B 0,C 180,E1 -1014.446,E2 -1014.446} C_VEL
LIN {X 0,Y 594.384,Z 307.44,A -85,B 0,C 180,E1 -1016.7,E2 -1016.7} C_VEL
LIN {X 0,Y 594.38,Z 307.441,A -85,B 0,C 180,E1 -1018.999,E2 -1018.999} C_VEL
LIN {X 0,Y 594.39,Z 307.449,A -85,B 0,C 180,E1 -1021.645,E2 -1021.645} C_VEL
LIN {X 0,Y 594.399,Z 307.438,A -85,B 0,C 180,E1 -1024.579,E2 -1024.579} C_VEL
LIN {X 0,Y 594.388,Z 307.45,A -85,B 0,C 180,E1 -1027.609,E2 -1027.609} C_VEL
LIN {X 0,Y 594.364,Z 307.443,A -85,B 0,C 180,E1 -1030.568,E2 -1030.568} C_VEL
LIN {X 0,Y 594.366,Z 307.448,A -85,B 0,C 180,E1 -1033.3,E2 -1033.3} C_VEL
LIN {X 0,Y 594.369,Z 307.444,A -85,B 0,C 180,E1 -1036.161,E2 -1036.161} C_VEL
LIN {X 0,Y 594.379,Z 307.441,A -85,B 0,C 180,E1 -1038.536,E2 -1038.536} C_VEL
LIN {X 0,Y 594.381,Z 307.447,A -85,B 0,C 180,E1 -1041.297,E2 -1041.297} C_VEL
LIN {X 0,Y 594.351,Z 307.45,A -85,B 0,C 180,E1 -1043.756,E2 -1043.756} C_VEL
LIN {X 0,Y 594.366,Z 307.443,A -85,B 0,C 180,E1 -1046.238,E2 -1046.238} C_VEL
LIN {X 0,Y 594.371,Z 307.442,A -85,B 0,C 180,E1 -1048.65,E2 -1048.65} C_VEL
LIN {X 0,Y 594.386,Z 307.444,A -85,B 0,C 180,E1 -1051.043,E2 -1051.043} C_VEL
LIN {X 0,Y 594.379,Z 307.442,A -85,B 0,C 180,E1 -1053.98,E2 -1053.98} C_VEL
LIN {X 0,Y 594.371,Z 307.442,A -85,B 0,C 180,E1 -1056.296,E2 -1056.296} C_VEL
LIN {X 0,Y 594.381,Z 307.444,A -85,B 0,C 180,E1 -1058.88,E2 -1058.88} C_VEL
LIN {X 0,Y 594.731,Z 308.866,A -85,B 0,C 180,E1 -1058.913,E2 -1058.913} C_VEL
LIN {X 0,Y 594.649,Z 400.984,A -85,B 0,C 180,E1 -1060.046,E2 -1060.046} C_VEL
LIN {X 0,Y 594.643,Z 413.972,A -85,B 0,C 180,E1 -1060.339,E2 -1060.339} C_VEL
LIN {X 0,Y 594.579,Z 427.519,A -85,B 0,C 180,E1 -1060.8,E2 -1060.8} C_VEL
LIN {X 0,Y 594.535,Z 438.267,A -85,B 0,C 180,E1 -1061.298,E2 -1061.298} C_VEL
LIN {X 0,Y 594.449,Z 448.945,A -85,B 0,C 180,E1 -1061.92,E2 -1061.92} C_VEL
LIN {X 0,Y 594.428,Z 458.81,A -85,B 0,C 180,E1 -1062.631,E2 -1062.631} C_VEL
LIN {X 0,Y 594.368,Z 468.787,A -85,B 0,C 180,E1 -1063.514,E2 -1063.514} C_VEL
LIN {X 0,Y 594.348,Z 476.914,A -85,B 0,C 180,E1 -1064.395,E2 -1064.395} C_VEL
LIN {X 0,Y 594.298,Z 484.759,A -85,B 0,C 180,E1 -1065.446,E2 -1065.446} C_VEL
LIN {X 0,Y 594.288,Z 490.088,A -85,B 0,C 180,E1 -1066.319,E2 -1066.319} C_VEL
LIN {X 0,Y 594.259,Z 495.21,A -85,B 0,C 180,E1 -1067.362,E2 -1067.362} C_VEL
LIN {X 0,Y 594.248,Z 499.153,A -85,B 0,C 180,E1 -1068.402,E2 -1068.402} C_VEL
LIN {X 0,Y 594.242,Z 501.188,A -85,B 0,C 180,E1 -1069.093,E2 -1069.093} C_VEL
LIN {X 0,Y 594.23,Z 502.765,A -85,B 0,C 180,E1 -1069.782,E2 -1069.782} C_VEL
LIN {X 0,Y 594.256,Z 503.91,A -85,B 0,C 180,E1 -1070.47,E2 -1070.47} C_VEL
LIN {X 0,Y 594.228,Z 504.64,A -85,B 0,C 180,E1 -1071.156,E2 -1071.156} C_VEL
LIN {X 0,Y 594.228,Z 504.959,A -85,B 0,C 180,E1 -1071.841,E2 -1071.841} C_VEL
LIN {X 0,Y 594.248,Z 504.881,A -85,B 0,C 180,E1 -1072.525,E2 -1072.525} C_VEL
LIN {X 0,Y 594.264,Z 504.153,A -85,B 0,C 180,E1 -1073.426,E2 -1073.426} C_VEL
LIN {X 0,Y 594.263,Z 502.21,A -85,B 0,C 180,E1 -1074.571,E2 -1074.571} C_VEL
LIN {X 0,Y 594.27,Z 499.458,A -85,B 0,C 180,E1 -1075.592,E2 -1075.592} C_VEL
LIN {X 0,Y 594.271,Z 495.7,A -85,B 0,C 180,E1 -1076.61,E2 -1076.61} C_VEL
LIN {X 0,Y 594.278,Z 490.849,A -85,B 0,C 180,E1 -1077.628,E2 -1077.628} C_VEL
LIN {X 0,Y 594.326,Z 483.626,A -85,B 0,C 180,E1 -1078.815,E2 -1078.815} C_VEL
LIN {X 0,Y 594.341,Z 475.737,A -85,B 0,C 180,E1 -1079.831,E2 -1079.831} C_VEL
LIN {X 0,Y 594.377,Z 467.729,A -85,B 0,C 180,E1 -1080.678,E2 -1080.678} C_VEL
LIN {X 0,Y 594.43,Z 457.976,A -85,B 0,C 180,E1 -1081.525,E2 -1081.525} C_VEL
LIN {X 0,Y 594.459,Z 447.14,A -85,B 0,C 180,E1 -1082.287,E2 -1082.287} C_VEL
LIN {X 0,Y 594.556,Z 434.83,A -85,B 0,C 180,E1 -1082.965,E2 -1082.965} C_VEL
LIN {X 0,Y 594.574,Z 422.696,A -85,B 0,C 180,E1 -1083.473,E2 -1083.473} C_VEL
LIN {X 0,Y 594.603,Z 410.886,A -85,B 0,C 180,E1 -1083.834,E2 -1083.834} C_VEL
LIN {X 0,Y 594.632,Z 398.247,A -85,B 0,C 180,E1 -1084.088,E2 -1084.088} C_VEL
LIN {X 0,Y 594.676,Z 308.812,A -85,B 0,C 180,E1 -1085.178,E2 -1085.178} C_VEL
LIN {X 0,Y 594.366,Z 307.446,A -85,B 0,C 180,E1 -1085.216,E2 -1085.216} C_VEL
LIN {X 0,Y 594.342,Z 307.446,A -85,B 0,C 180,E1 -1087.474,E2 -1087.474} C_VEL
LIN {X 0,Y 594.321,Z 307.449,A -85,B 0,C 180,E1 -1089.53,E2 -1089.53} C_VEL
LIN {X 0,Y 594.37,Z 307.448,A -85,B 0,C 180,E1 -1092.289,E2 -1092.289} C_VEL
LIN {X 0,Y 594.338,Z 307.448,A -85,B 0,C 180,E1 -1095.079,E2 -1095.079} C_VEL
LIN {X 0,Y 594.319,Z 307.449,A -85,B 0,C 180,E1 -1097.196,E2 -1097.196} C_VEL
LIN {X 0,Y 594.336,Z 307.447,A -85,B 0,C 180,E1 -1099.336,E2 -1099.336} C_VEL
LIN {X 0,Y 594.326,Z 307.448,A -85,B 0,C 180,E1 -1101.505,E2 -1101.505} C_VEL
LIN {X 0,Y 594.349,Z 307.446,A -85,B 0,C 180,E1 -1103.706,E2 -1103.706} C_VEL
LIN {X 0,Y 594.34,Z 307.449,A -85,B 0,C 180,E1 -1106.702,E2 -1106.702} C_VEL
LIN {X 0,Y 594.35,Z 307.448,A -85,B 0,C 180,E1 -1109.778,E2 -1109.778} C_VEL
LIN {X 0,Y 594.358,Z 307.454,A -85,B 0,C 180,E1 -1112.148,E2 -1112.148} C_VEL
LIN {X 0,Y 594.355,Z 307.446,A -85,B 0,C 180,E1 -1114.582,E2 -1114.582} C_VEL
LIN {X 0,Y 594.361,Z 307.447,A -85,B 0,C 180,E1 -1117.604,E2 -1117.604} C_VEL
LIN {X 0,Y 594.359,Z 307.444,A -85,B 0,C 180,E1 -1120.568,E2 -1120.568} C_VEL
LIN {X 0,Y 594.347,Z 307.447,A -85,B 0,C 180,E1 -1123.302,E2 -1123.302} C_VEL
LIN {X 0,Y 594.349,Z 307.449,A -85,B 0,C 180,E1 -1126.163,E2 -1126.163} C_VEL
LIN {X 0,Y 594.372,Z 307.442,A -85,B 0,C 180,E1 -1128.535,E2 -1128.535} C_VEL
LIN {X 0,Y 594.371,Z 307.446,A -85,B 0,C 180,E1 -1131.298,E2 -1131.298} C_VEL
LIN {X 0,Y 594.352,Z 307.453,A -85,B 0,C 180,E1 -1133.755,E2 -1133.755} C_VEL
LIN {X 0,Y 594.366,Z 307.444,A -85,B 0,C 180,E1 -1136.238,E2 -1136.238} C_VEL
LIN {X 0,Y 594.368,Z 307.442,A -85,B 0,C 180,E1 -1138.649,E2 -1138.649} C_VEL
LIN {X 0,Y 594.382,Z 307.444,A -85,B 0,C 180,E1 -1141.043,E2 -1141.043} C_VEL
LIN {X 0,Y 594.375,Z 307.543,A -85,B 0,C 180,E1 -1143.925,E2 -1143.925} C_VEL
LIN {X 0,Y 595.12,Z 311.884,A -85,B 0,C 180,E1 -1144.466,E2 -1144.466} C_VEL
LIN {X 0,Y 594.952,Z 336.26,A -85,B 0,C 180,E1 -1147.264,E2 -1147.264} C_VEL
LIN {X 0,Y 594.805,Z 361.817,A -85,B 0,C 180,E1 -1150.141,E2 -1150.141} C_VEL
LIN {X 0,Y 594.633,Z 388.613,A -85,B 0,C 180,E1 -1153.103,E2 -1153.103} C_VEL
LIN {X 0,Y 594.529,Z 417.068,A -85,B 0,C 180,E1 -1156.203,E2 -1156.203} C_VEL
LIN {X 0,Y 594.509,Z 421.336,A -85,B 0,C 180,E1 -1156.65,E2 -1156.65} C_VEL
LIN {X 0,Y 594.785,Z 430.28,A -85,B 0,C 180,E1 -1156.765,E2 -1156.765} C_VEL
LIN {X 0,Y 594.656,Z 530.936,A -85,B 0,C 180,E1 -1157.999,E2 -1157.999} C_VEL
LIN {X 0,Y 594.617,Z 544.211,A -85,B 0,C 180,E1 -1158.3,E2 -1158.3} C_VEL
LIN {X 0,Y 594.564,Z 556.413,A -85,B 0,C 180,E1 -1158.712,E2 -1158.712} C_VEL
LIN {X 0,Y 594.538,Z 568.629,A -85,B 0,C 180,E1 -1159.27,E2 -1159.27} C_VEL
LIN {X 0,Y 594.469,Z 580.197,A -85,B 0,C 180,E1 -1159.957,E2 -1159.957} C_VEL
LIN {X 0,Y 594.413,Z 590.594,A -85,B 0,C 180,E1 -1160.729,E2 -1160.729} C_VEL
LIN {X 0,Y 594.383,Z 599.11,A -85,B 0,C 180,E1 -1161.5,E2 -1161.5} C_VEL
LIN {X 0,Y 594.347,Z 606.959,A -85,B 0,C 180,E1 -1162.355,E2 -1162.355} C_VEL
LIN {X 0,Y 594.283,Z 614.813,A -85,B 0,C 180,E1 -1163.408,E2 -1163.408} C_VEL
LIN {X 0,Y 594.289,Z 621.68,A -85,B 0,C 180,E1 -1164.571,E2 -1164.571} C_VEL
LIN {X 0,Y 594.27,Z 626.371,A -85,B 0,C 180,E1 -1165.591,E2 -1165.591} C_VEL
LIN {X 0,Y 594.267,Z 629.956,A -85,B 0,C 180,E1 -1166.61,E2 -1166.61} C_VEL
LIN {X 0,Y 594.226,Z 631.808,A -85,B 0,C 180,E1 -1167.288,E2 -1167.288} C_VEL
LIN {X 0,Y 594.24,Z 633.201,A -85,B 0,C 180,E1 -1167.967,E2 -1167.967} C_VEL
LIN {X 0,Y 594.239,Z 634.784,A -85,B 0,C 180,E1 -1169.322,E2 -1169.322} C_VEL
LIN {X 0,Y 594.236,Z 635,A -85,B 0,C 180,E1 -1170,E2 -1170} C_VEL
LIN {X 0,Y 594.247,Z 634.185,A -85,B 0,C 180,E1 -1171.355,E2 -1171.355} C_VEL
LIN {X 0,Y 594.24,Z 633.202,A -85,B 0,C 180,E1 -1172.033,E2 -1172.033} C_VEL
LIN {X 0,Y 594.226,Z 631.81,A -85,B 0,C 180,E1 -1172.711,E2 -1172.711} C_VEL
LIN {X 0,Y 594.288,Z 628.896,A -85,B 0,C 180,E1 -1173.729,E2 -1173.729} C_VEL
LIN {X 0,Y 594.242,Z 624.95,A -85,B 0,C 180,E1 -1174.749,E2 -1174.749} C_VEL
LIN {X 0,Y 594.304,Z 618.878,A -85,B 0,C 180,E1 -1175.939,E2 -1175.939} C_VEL
LIN {X 0,Y 594.308,Z 612.237,A -85,B 0,C 180,E1 -1176.962,E2 -1176.962} C_VEL
LIN {X 0,Y 594.359,Z 603.99,A -85,B 0,C 180,E1 -1177.986,E2 -1177.986} C_VEL
LIN {X 0,Y 594.382,Z 595.538,A -85,B 0,C 180,E1 -1178.842,E2 -1178.842} C_VEL
LIN {X 0,Y 594.427,Z 585.094,A -85,B 0,C 180,E1 -1179.699,E2 -1179.699} C_VEL
LIN {X 0,Y 594.482,Z 574.76,A -85,B 0,C 180,E1 -1180.386,E2 -1180.386} C_VEL
LIN {X 0,Y 594.559,Z 563.708,A -85,B 0,C 180,E1 -1180.974,E2 -1180.974} C_VEL
LIN {X 0,Y 594.583,Z 551.707,A -85,B 0,C 180,E1 -1181.464,E2 -1181.464} C_VEL
LIN {X 0,Y 594.636,Z 538.352,A -85,B 0,C 180,E1 -1181.85,E2 -1181.85} C_VEL
LIN {X 0,Y 594.692,Z 525.086,A -85,B 0,C 180,E1 -1182.087,E2 -1182.087} C_VEL
LIN {X 0,Y 594.628,Z 422.026,A -85,B 0,C 180,E1 -1183.339,E2 -1183.339} C_VEL
LIN {X 0,Y 594.507,Z 421.014,A -85,B 0,C 180,E1 -1183.371,E2 -1183.371} C_VEL
LIN {X 0,Y 594.598,Z 395.645,A -85,B 0,C 180,E1 -1186.127,E2 -1186.127} C_VEL
LIN {X 0,Y 594.744,Z 370.447,A -85,B 0,C 180,E1 -1188.9,E2 -1188.9} C_VEL
LIN {X 0,Y 594.884,Z 345.712,A -85,B 0,C 180,E1 -1191.666,E2 -1191.666} C_VEL
LIN {X 0,Y 595.062,Z 321.551,A -85,B 0,C 180,E1 -1194.417,E2 -1194.417} C_VEL
LIN {X 0,Y 594.993,Z 310.276,A -85,B 0,C 180,E1 -1195.727,E2 -1195.727} C_VEL
LIN {X 0,Y 594.369,Z 307.45,A -85,B 0,C 180,E1 -1196.089,E2 -1196.089} C_VEL
LIN {X 0,Y 594.38,Z 307.444,A -85,B 0,C 180,E1 -1198.999,E2 -1198.999} C_VEL
LIN {X 0,Y 594.378,Z 307.442,A -85,B 0,C 180,E1 -1201.642,E2 -1201.642} C_VEL
LIN {X 0,Y 594.368,Z 307.449,A -85,B 0,C 180,E1 -1204.581,E2 -1204.581} C_VEL
LIN {X 0,Y 594.388,Z 307.441,A -85,B 0,C 180,E1 -1207.608,E2 -1207.608} C_VEL
LIN {X 0,Y 594.361,Z 307.448,A -85,B 0,C 180,E1 -1210.568,E2 -1210.568} C_VEL
LIN {X 0,Y 594.346,Z 307.445,A -85,B 0,C 180,E1 -1213.302,E2 -1213.302} C_VEL
LIN {X 0,Y 594.346,Z 307.455,A -85,B 0,C 180,E1 -1216.163,E2 -1216.163} C_VEL
LIN {X 0,Y 594.366,Z 307.446,A -85,B 0,C 180,E1 -1218.534,E2 -1218.534} C_VEL
LIN {X 0,Y 594.365,Z 307.443,A -85,B 0,C 180,E1 -1221.298,E2 -1221.298} C_VEL
LIN {X 0,Y 594.345,Z 307.452,A -85,B 0,C 180,E1 -1223.755,E2 -1223.755} C_VEL
LIN {X 0,Y 594.345,Z 307.45,A -85,B 0,C 180,E1 -1226.236,E2 -1226.236} C_VEL
LIN {X 0,Y 594.326,Z 307.448,A -85,B 0,C 180,E1 -1228.647,E2 -1228.647} C_VEL
LIN {X 0,Y 594.34,Z 307.447,A -85,B 0,C 180,E1 -1231.05,E2 -1231.05} C_VEL
LIN {X 0,Y 594.341,Z 307.451,A -85,B 0,C 180,E1 -1234.054,E2 -1234.054} C_VEL
LIN {X 0,Y 594.347,Z 307.447,A -85,B 0,C 180,E1 -1236.294,E2 -1236.294} C_VEL
LIN {X 0,Y 594.368,Z 307.447,A -85,B 0,C 180,E1 -1239.223,E2 -1239.223} C_VEL
LIN {X 0,Y 594.314,Z 307.451,A -85,B 0,C 180,E1 -1242.093,E2 -1242.093} C_VEL
LIN {X 0,Y 594.33,Z 307.448,A -85,B 0,C 180,E1 -1244.218,E2 -1244.218} C_VEL
LIN {X 0,Y 594.341,Z 307.45,A -85,B 0,C 180,E1 -1247.016,E2 -1247.016} C_VEL
LIN {X 0,Y 594.374,Z 307.445,A -85,B 0,C 180,E1 -1248.884,E2 -1248.884} C_VEL
LIN {X 0,Y 594.738,Z 311.79,A -85,B 0,C 180,E1 -1248.949,E2 -1248.949} C_VEL
LIN {X 0,Y 594.603,Z 401.09,A -85,B 0,C 180,E1 -1250.045,E2 -1250.045} C_VEL
LIN {X 0,Y 594.571,Z 414.258,A -85,B 0,C 180,E1 -1250.346,E2 -1250.346} C_VEL
LIN {X 0,Y 594.567,Z 427.939,A -85,B 0,C 180,E1 -1250.817,E2 -1250.817} C_VEL
LIN {X 0,Y 594.538,Z 438.89,A -85,B 0,C 180,E1 -1251.331,E2 -1251.331} C_VEL
LIN {X 0,Y 594.437,Z 450.364,A -85,B 0,C 180,E1 -1252.014,E2 -1252.014} C_VEL
LIN {X 0,Y 594.435,Z 460.687,A -85,B 0,C 180,E1 -1252.783,E2 -1252.783} C_VEL
LIN {X 0,Y 594.37,Z 470.891,A -85,B 0,C 180,E1 -1253.727,E2 -1253.727} C_VEL
LIN {X 0,Y 594.32,Z 479.684,A -85,B 0,C 180,E1 -1254.741,E2 -1254.741} C_VEL
LIN {X 0,Y 594.276,Z 486.8,A -85,B 0,C 180,E1 -1255.761,E2 -1255.761} C_VEL
LIN {X 0,Y 594.275,Z 491.634,A -85,B 0,C 180,E1 -1256.61,E2 -1256.61} C_VEL
LIN {X 0,Y 594.275,Z 496.318,A -85,B 0,C 180,E1 -1257.627,E2 -1257.627} C_VEL
LIN {X 0,Y 594.253,Z 499.912,A -85,B 0,C 180,E1 -1258.644,E2 -1258.644} C_VEL
LIN {X 0,Y 594.24,Z 501.771,A -85,B 0,C 180,E1 -1259.322,E2 -1259.322} C_VEL
LIN {X 0,Y 594.236,Z 503.185,A -85,B 0,C 180,E1 -1260,E2 -1260} C_VEL
LIN {X 0,Y 594.247,Z 504.776,A -85,B 0,C 180,E1 -1261.355,E2 -1261.355} C_VEL
LIN {X 0,Y 594.24,Z 505,A -85,B 0,C 180,E1 -1262.033,E2 -1262.033} C_VEL
LIN {X 0,Y 594.258,Z 504.194,A -85,B 0,C 180,E1 -1263.39,E2 -1263.39} C_VEL
LIN {X 0,Y 594.255,Z 503.219,A -85,B 0,C 180,E1 -1264.069,E2 -1264.069} C_VEL
LIN {X 0,Y 594.23,Z 501.813,A -85,B 0,C 180,E1 -1264.749,E2 -1264.749} C_VEL
LIN {X 0,Y 594.266,Z 498.896,A -85,B 0,C 180,E1 -1265.769,E2 -1265.769} C_VEL
LIN {X 0,Y 594.277,Z 494.944,A -85,B 0,C 180,E1 -1266.791,E2 -1266.791} C_VEL
LIN {X 0,Y 594.305,Z 489.848,A -85,B 0,C 180,E1 -1267.816,E2 -1267.816} C_VEL
LIN {X 0,Y 594.313,Z 482.185,A -85,B 0,C 180,E1 -1269.014,E2 -1269.014} C_VEL
LIN {X 0,Y 594.344,Z 473.857,A -85,B 0,C 180,E1 -1270.044,E2 -1270.044} C_VEL
LIN {X 0,Y 594.391,Z 465.317,A -85,B 0,C 180,E1 -1270.905,E2 -1270.905} C_VEL
LIN {X 0,Y 594.46,Z 454.786,A -85,B 0,C 180,E1 -1271.767,E2 -1271.767} C_VEL
LIN {X 0,Y 594.499,Z 444.31,A -85,B 0,C 180,E1 -1272.459,E2 -1272.459} C_VEL
LIN {X 0,Y 594.555,Z 434.567,A -85,B 0,C 180,E1 -1272.978,E2 -1272.978} C_VEL
LIN {X 0,Y 593.916,Z 429.311,A -85,B 0,C 180,E1 -1273.233,E2 -1273.233} C_VEL
LIN {X 0,Y 591.08,Z 420.674,A -85,B 0,C 180,E1 -1273.621,E2 -1273.621} C_VEL
LIN {X 0,Y 588.296,Z 411.772,A -85,B 0,C 180,E1 -1273.942,E2 -1273.942} C_VEL
LIN {X 0,Y 587.728,Z 406.11,A -85,B 0,C 180,E1 -1274.09,E2 -1274.09} C_VEL
LIN {X 0,Y 587.732,Z 392.196,A -85,B 0,C 180,E1 -1274.313,E2 -1274.313} C_VEL
LIN {X 0,Y 587.774,Z 309.991,A -85,B 0,C 180,E1 -1275.321,E2 -1275.321} C_VEL
LIN {X 0,Y 587.343,Z 308.333,A -85,B 0,C 180,E1 -1275.351,E2 -1275.351} C_VEL
LIN {X 0,Y 587.348,Z 308.318,A -85,B 0,C 180,E1 -1277.406,E2 -1277.406} C_VEL
LIN {X 0,Y 587.326,Z 308.324,A -85,B 0,C 180,E1 -1280.305,E2 -1280.305} C_VEL
LIN {X 0,Y 587.313,Z 308.323,A -85,B 0,C 180,E1 -1283.259,E2 -1283.259} C_VEL
LIN {X 0,Y 587.329,Z 308.319,A -85,B 0,C 180,E1 -1285.517,E2 -1285.517} C_VEL
LIN {X 0,Y 587.341,Z 308.318,A -85,B 0,C 180,E1 -1287.818,E2 -1287.818} C_VEL
LIN {X 0,Y 587.326,Z 308.328,A -85,B 0,C 180,E1 -1290.508,E2 -1290.508} C_VEL
LIN {X 0,Y 587.337,Z 308.32,A -85,B 0,C 180,E1 -1293.111,E2 -1293.111} C_VEL
LIN {X 0,Y 587.29,Z 308.325,A -85,B 0,C 180,E1 -1295.9,E2 -1295.9} C_VEL
LIN {X 0,Y 587.325,Z 308.329,A -85,B 0,C 180,E1 -1298.479,E2 -1298.479} C_VEL
LIN {X 0,Y 587.335,Z 308.319,A -85,B 0,C 180,E1 -1301.157,E2 -1301.157} C_VEL
LIN {X 0,Y 587.326,Z 308.324,A -85,B 0,C 180,E1 -1304.113,E2 -1304.113} C_VEL
LIN {X 0,Y 587.311,Z 308.323,A -85,B 0,C 180,E1 -1306.993,E2 -1306.993} C_VEL
LIN {X 0,Y 587.314,Z 308.322,A -85,B 0,C 180,E1 -1309.745,E2 -1309.745} C_VEL
LIN {X 0,Y 587.342,Z 308.328,A -85,B 0,C 180,E1 -1312.392,E2 -1312.392} C_VEL
LIN {X 0,Y 587.351,Z 308.318,A -85,B 0,C 180,E1 -1314.946,E2 -1314.946} C_VEL
LIN {X 0,Y 587.336,Z 308.318,A -85,B 0,C 180,E1 -1317.421,E2 -1317.421} C_VEL
LIN {X 0,Y 587.333,Z 308.321,A -85,B 0,C 180,E1 -1319.83,E2 -1319.83} C_VEL
LIN {X 0,Y 587.35,Z 308.327,A -85,B 0,C 180,E1 -1322.307,E2 -1322.307} C_VEL
LIN {X 0,Y 587.336,Z 308.325,A -85,B 0,C 180,E1 -1324.483,E2 -1324.483} C_VEL
LIN {X 0,Y 587.337,Z 308.319,A -85,B 0,C 180,E1 -1327.486,E2 -1327.486} C_VEL
LIN {X 0,Y 587.339,Z 308.324,A -85,B 0,C 180,E1 -1330.425,E2 -1330.425} C_VEL
LIN {X 0,Y 587.344,Z 308.317,A -85,B 0,C 180,E1 -1333.311,E2 -1333.311} C_VEL
LIN {X 0,Y 587.359,Z 308.326,A -85,B 0,C 180,E1 -1336.154,E2 -1336.154} C_VEL
LIN {X 0,Y 587.339,Z 308.318,A -85,B 0,C 180,E1 -1338.962,E2 -1338.962} C_VEL
LIN {X 0,Y 587.363,Z 308.319,A -85,B 0,C 180,E1 -1341.745,E2 -1341.745} C_VEL
LIN {X 0,Y 587.357,Z 308.319,A -85,B 0,C 180,E1 -1344.507,E2 -1344.507} C_VEL
LIN {X 0,Y 587.369,Z 308.315,A -85,B 0,C 180,E1 -1347.257,E2 -1347.257} C_VEL
LIN {X 0,Y 587.383,Z 308.322,A -85,B 0,C 180,E1 -1350,E2 -1350} C_VEL
LIN {X 0,Y 587.368,Z 308.315,A -85,B 0,C 180,E1 -1352.743,E2 -1352.743} C_VEL
LIN {X 0,Y 587.357,Z 308.319,A -85,B 0,C 180,E1 -1355.493,E2 -1355.493} C_VEL
LIN {X 0,Y 587.363,Z 308.32,A -85,B 0,C 180,E1 -1358.255,E2 -1358.255} C_VEL
LIN {X 0,Y 587.346,Z 308.317,A -85,B 0,C 180,E1 -1361.134,E2 -1361.134} C_VEL
LIN {X 0,Y 587.364,Z 308.319,A -85,B 0,C 180,E1 -1364.261,E2 -1364.261} C_VEL
LIN {X 0,Y 587.355,Z 308.319,A -85,B 0,C 180,E1 -1367.406,E2 -1367.406} C_VEL
LIN {X 0,Y 587.326,Z 308.322,A -85,B 0,C 180,E1 -1370.305,E2 -1370.305} C_VEL
LIN {X 0,Y 587.321,Z 308.322,A -85,B 0,C 180,E1 -1373.259,E2 -1373.259} C_VEL
LIN {X 0,Y 587.336,Z 308.324,A -85,B 0,C 180,E1 -1375.517,E2 -1375.517} C_VEL
LIN {X 0,Y 587.347,Z 308.326,A -85,B 0,C 180,E1 -1377.818,E2 -1377.818} C_VEL
LIN {X 0,Y 587.341,Z 308.318,A -85,B 0,C 180,E1 -1380.511,E2 -1380.511} C_VEL
LIN {X 0,Y 587.334,Z 308.324,A -85,B 0,C 180,E1 -1383.397,E2 -1383.397} C_VEL
LIN {X 0,Y 587.303,Z 308.329,A -85,B 0,C 180,E1 -1385.9,E2 -1385.9} C_VEL
LIN {X 0,Y 587.33,Z 308.319,A -85,B 0,C 180,E1 -1388.48,E2 -1388.48} C_VEL
LIN {X 0,Y 587.335,Z 308.321,A -85,B 0,C 180,E1 -1391.157,E2 -1391.157} C_VEL
LIN {X 0,Y 587.312,Z 308.324,A -85,B 0,C 180,E1 -1394.112,E2 -1394.112} C_VEL
LIN {X 0,Y 587.317,Z 308.323,A -85,B 0,C 180,E1 -1396.994,E2 -1396.994} C_VEL
LIN {X 0,Y 587.312,Z 308.328,A -85,B 0,C 180,E1 -1399.746,E2 -1399.746} C_VEL
LIN {X 0,Y 587.344,Z 308.317,A -85,B 0,C 180,E1 -1402.393,E2 -1402.393} C_VEL
LIN {X 0,Y 587.344,Z 308.325,A -85,B 0,C 180,E1 -1405.654,E2 -1405.654} C_VEL
LIN {X 0,Y 587.342,Z 308.318,A -85,B 0,C 180,E1 -1408.232,E2 -1408.232} C_VEL
LIN {X 0,Y 587.351,Z 308.318,A -85,B 0,C 180,E1 -1410.867,E2 -1410.867} C_VEL
LIN {X 0,Y 587.34,Z 308.321,A -85,B 0,C 180,E1 -1413.824,E2 -1413.824} C_VEL
LIN {X 0,Y 587.318,Z 308.322,A -85,B 0,C 180,E1 -1415.993,E2 -1415.993} C_VEL
LIN {X 0,Y 587.357,Z 308.318,A -85,B 0,C 180,E1 -1418.729,E2 -1418.729} C_VEL
LIN {X 0,Y 587.789,Z 309.996,A -85,B 0,C 180,E1 -1418.769,E2 -1418.769} C_VEL
LIN {X 0,Y 587.717,Z 400.279,A -85,B 0,C 180,E1 -1419.892,E2 -1419.892} C_VEL
LIN {X 0,Y 587.687,Z 412.765,A -85,B 0,C 180,E1 -1420.164,E2 -1420.164} C_VEL
LIN {X 0,Y 587.599,Z 425.686,A -85,B 0,C 180,E1 -1420.592,E2 -1420.592} C_VEL
LIN {X 0,Y 587.551,Z 438.07,A -85,B 0,C 180,E1 -1421.158,E2 -1421.158} C_VEL
LIN {X 0,Y 587.451,Z 448.766,A -85,B 0,C 180,E1 -1421.788,E2 -1421.788} C_VEL
LIN {X 0,Y 587.412,Z 458.66,A -85,B 0,C 180,E1 -1422.506,E2 -1422.506} C_VEL
LIN {X 0,Y 587.328,Z 467.759,A -85,B 0,C 180,E1 -1423.311,E2 -1423.311} C_VEL
LIN {X 0,Y 587.281,Z 477.54,A -85,B 0,C 180,E1 -1424.38,E2 -1424.38} C_VEL
LIN {X 0,Y 587.221,Z 485.261,A -85,B 0,C 180,E1 -1425.444,E2 -1425.444} C_VEL
LIN {X 0,Y 587.198,Z 491.415,A -85,B 0,C 180,E1 -1426.504,E2 -1426.504} C_VEL
LIN {X 0,Y 587.181,Z 496.248,A -85,B 0,C 180,E1 -1427.559,E2 -1427.559} C_VEL
LIN {X 0,Y 587.15,Z 499.928,A -85,B 0,C 180,E1 -1428.61,E2 -1428.61} C_VEL
LIN {X 0,Y 587.139,Z 502.56,A -85,B 0,C 180,E1 -1429.657,E2 -1429.657} C_VEL
LIN {X 0,Y 587.151,Z 503.773,A -85,B 0,C 180,E1 -1430.353,E2 -1430.353} C_VEL
LIN {X 0,Y 587.128,Z 504.575,A -85,B 0,C 180,E1 -1431.048,E2 -1431.048} C_VEL
LIN {X 0,Y 587.146,Z 504.914,A -85,B 0,C 180,E1 -1432.434,E2 -1432.434} C_VEL
LIN {X 0,Y 587.189,Z 504.171,A -85,B 0,C 180,E1 -1433.426,E2 -1433.426} C_VEL
LIN {X 0,Y 587.18,Z 502.408,A -85,B 0,C 180,E1 -1434.506,E2 -1434.506} C_VEL
LIN {X 0,Y 587.186,Z 499.75,A -85,B 0,C 180,E1 -1435.538,E2 -1435.538} C_VEL
LIN {X 0,Y 587.197,Z 496.089,A -85,B 0,C 180,E1 -1436.569,E2 -1436.569} C_VEL
LIN {X 0,Y 587.193,Z 491.348,A -85,B 0,C 180,E1 -1437.599,E2 -1437.599} C_VEL
LIN {X 0,Y 587.207,Z 485.375,A -85,B 0,C 180,E1 -1438.629,E2 -1438.629} C_VEL
LIN {X 0,Y 587.271,Z 477.952,A -85,B 0,C 180,E1 -1439.657,E2 -1439.657} C_VEL
LIN {X 0,Y 587.324,Z 468.714,A -85,B 0,C 180,E1 -1440.686,E2 -1440.686} C_VEL
LIN {X 0,Y 587.393,Z 459.174,A -85,B 0,C 180,E1 -1441.543,E2 -1441.543} C_VEL
LIN {X 0,Y 587.43,Z 449.881,A -85,B 0,C 180,E1 -1442.229,E2 -1442.229} C_VEL
LIN {X 0,Y 587.518,Z 439.956,A -85,B 0,C 180,E1 -1442.829,E2 -1442.829} C_VEL
LIN {X 0,Y 587.572,Z 429.376,A -85,B 0,C 180,E1 -1443.343,E2 -1443.343} C_VEL
LIN {X 0,Y 587.616,Z 416.678,A -85,B 0,C 180,E1 -1443.815,E2 -1443.815} C_VEL
LIN {X 0,Y 587.666,Z 402.699,A -85,B 0,C 180,E1 -1444.158,E2 -1444.158} C_VEL
LIN {X 0,Y 587.728,Z 375.093,A -85,B 0,C 180,E1 -1444.523,E2 -1444.523} C_VEL
LIN {X 0,Y 587.728,Z 309.9,A -85,B 0,C 180,E1 -1445.323,E2 -1445.323} C_VEL
LIN {X 0,Y 587.315,Z 308.323,A -85,B 0,C 180,E1 -1445.365,E2 -1445.365} C_VEL
LIN {X 0,Y 587.304,Z 308.323,A -85,B 0,C 180,E1 -1447.564,E2 -1447.564} C_VEL
LIN {X 0,Y 587.293,Z 308.331,A -85,B 0,C 180,E1 -1450.341,E2 -1450.341} C_VEL
LIN {X 0,Y 587.287,Z 308.326,A -85,B 0,C 180,E1 -1453.143,E2 -1453.143} C_VEL
LIN {X 0,Y 587.299,Z 308.324,A -85,B 0,C 180,E1 -1455.264,E2 -1455.264} C_VEL
LIN {X 0,Y 587.267,Z 308.327,A -85,B 0,C 180,E1 -1457.409,E2 -1457.409} C_VEL
LIN {X 0,Y 587.287,Z 308.325,A -85,B 0,C 180,E1 -1459.577,E2 -1459.577} C_VEL
LIN {X 0,Y 587.306,Z 308.329,A -85,B 0,C 180,E1 -1462.515,E2 -1462.515} C_VEL
LIN {X 0,Y 587.298,Z 308.326,A -85,B 0,C 180,E1 -1464.761,E2 -1464.761} C_VEL
LIN {X 0,Y 587.29,Z 308.326,A -85,B 0,C 180,E1 -1467.68,E2 -1467.68} C_VEL
LIN {X 0,Y 587.317,Z 308.325,A -85,B 0,C 180,E1 -1470.506,E2 -1470.506} C_VEL
LIN {X 0,Y 587.324,Z 308.321,A -85,B 0,C 180,E1 -1473.398,E2 -1473.398} C_VEL
LIN {X 0,Y 587.278,Z 308.333,A -85,B 0,C 180,E1 -1475.901,E2 -1475.901} C_VEL
LIN {X 0,Y 587.316,Z 308.323,A -85,B 0,C 180,E1 -1478.481,E2 -1478.481} C_VEL
LIN {X 0,Y 587.309,Z 308.322,A -85,B 0,C 180,E1 -1481.16,E2 -1481.16} C_VEL
LIN {X 0,Y 587.307,Z 308.328,A -85,B 0,C 180,E1 -1484.111,E2 -1484.111} C_VEL
LIN {X 0,Y 587.291,Z 308.324,A -85,B 0,C 180,E1 -1486.991,E2 -1486.991} C_VEL
LIN {X 0,Y 587.309,Z 308.332,A -85,B 0,C 180,E1 -1489.745,E2 -1489.745} C_VEL
LIN {X 0,Y 587.324,Z 308.321,A -85,B 0,C 180,E1 -1492.39,E2 -1492.39} C_VEL
LIN {X 0,Y 587.339,Z 308.328,A -85,B 0,C 180,E1 -1495.654,E2 -1495.654} C_VEL
LIN {X 0,Y 587.343,Z 308.319,A -85,B 0,C 180,E1 -1498.231,E2 -1498.231} C_VEL
LIN {X 0,Y 587.35,Z 308.319,A -85,B 0,C 180,E1 -1500.867,E2 -1500.867} C_VEL
LIN {X 0,Y 587.357,Z 308.46,A -85,B 0,C 180,E1 -1503.722,E2 -1503.722} C_VEL
LIN {X 0,Y 588.349,Z 313.495,A -85,B 0,C 180,E1 -1504.341,E2 -1504.341} C_VEL
LIN {X 0,Y 588.104,Z 338.569,A -85,B 0,C 180,E1 -1507.251,E2 -1507.251} C_VEL
LIN {X 0,Y 587.904,Z 363.428,A -85,B 0,C 180,E1 -1510.08,E2 -1510.08} C_VEL
LIN {X 0,Y 587.687,Z 390.238,A -85,B 0,C 180,E1 -1513.078,E2 -1513.078} C_VEL
LIN {X 0,Y 587.537,Z 418.193,A -85,B 0,C 180,E1 -1516.158,E2 -1516.158} C_VEL
LIN {X 0,Y 587.5,Z 421.336,A -85,B 0,C 180,E1 -1516.488,E2 -1516.488} C_VEL
LIN {X 0,Y 587.866,Z 426.702,A -85,B 0,C 180,E1 -1516.563,E2 -1516.563} C_VEL
LIN {X 0,Y 587.718,Z 530.936,A -85,B 0,C 180,E1 -1517.855,E2 -1517.855} C_VEL
LIN {X 0,Y 587.669,Z 544.212,A -85,B 0,C 180,E1 -1518.16,E2 -1518.16} C_VEL
LIN {X 0,Y 587.587,Z 556.67,A -85,B 0,C 180,E1 -1518.586,E2 -1518.586} C_VEL
LIN {X 0,Y 587.552,Z 568.627,A -85,B 0,C 180,E1 -1519.141,E2 -1519.141} C_VEL
LIN {X 0,Y 587.465,Z 580.199,A -85,B 0,C 180,E1 -1519.836,E2 -1519.836} C_VEL
LIN {X 0,Y 587.391,Z 590.596,A -85,B 0,C 180,E1 -1520.618,E2 -1520.618} C_VEL
LIN {X 0,Y 587.322,Z 599.11,A -85,B 0,C 180,E1 -1521.397,E2 -1521.397} C_VEL
LIN {X 0,Y 587.274,Z 606.959,A -85,B 0,C 180,E1 -1522.263,E2 -1522.263} C_VEL
LIN {X 0,Y 587.231,Z 613.468,A -85,B 0,C 180,E1 -1523.126,E2 -1523.126} C_VEL
LIN {X 0,Y 587.236,Z 619.866,A -85,B 0,C 180,E1 -1524.161,E2 -1524.161} C_VEL
LIN {X 0,Y 587.147,Z 624.949,A -85,B 0,C 180,E1 -1525.194,E2 -1525.194} C_VEL
LIN {X 0,Y 587.212,Z 628.895,A -85,B 0,C 180,E1 -1526.226,E2 -1526.226} C_VEL
LIN {X 0,Y 587.132,Z 631.808,A -85,B 0,C 180,E1 -1527.255,E2 -1527.255} C_VEL
LIN {X 0,Y 587.139,Z 633.2,A -85,B 0,C 180,E1 -1527.942,E2 -1527.942} C_VEL
LIN {X 0,Y 587.14,Z 634.784,A -85,B 0,C 180,E1 -1529.314,E2 -1529.314} C_VEL
LIN {X 0,Y 587.137,Z 635,A -85,B 0,C 180,E1 -1530,E2 -1530} C_VEL
LIN {X 0,Y 587.147,Z 634.185,A -85,B 0,C 180,E1 -1531.372,E2 -1531.372} C_VEL
LIN {X 0,Y 587.139,Z 633.201,A -85,B 0,C 180,E1 -1532.058,E2 -1532.058} C_VEL
LIN {X 0,Y 587.132,Z 631.81,A -85,B 0,C 180,E1 -1532.744,E2 -1532.744} C_VEL
LIN {X 0,Y 587.212,Z 628.896,A -85,B 0,C 180,E1 -1533.774,E2 -1533.774} C_VEL
LIN {X 0,Y 587.147,Z 624.95,A -85,B 0,C 180,E1 -1534.806,E2 -1534.806} C_VEL
LIN {X 0,Y 587.217,Z 618.878,A -85,B 0,C 180,E1 -1536.011,E2 -1536.011} C_VEL
LIN {X 0,Y 587.245,Z 612.237,A -85,B 0,C 180,E1 -1537.046,E2 -1537.046} C_VEL
LIN {X 0,Y 587.299,Z 603.99,A -85,B 0,C 180,E1 -1538.083,E2 -1538.083} C_VEL
LIN {X 0,Y 587.343,Z 595.538,A -85,B 0,C 180,E1 -1538.949,E2 -1538.949} C_VEL
LIN {X 0,Y 587.416,Z 585.096,A -85,B 0,C 180,E1 -1539.816,E2 -1539.816} C_VEL
LIN {X 0,Y 587.496,Z 574.758,A -85,B 0,C 180,E1 -1540.511,E2 -1540.511} C_VEL
LIN {X 0,Y 587.584,Z 562.808,A -85,B 0,C 180,E1 -1541.149,E2 -1541.149} C_VEL
LIN {X 0,Y 587.625,Z 550.595,A -85,B 0,C 180,E1 -1541.639,E2 -1541.639} C_VEL
LIN {X 0,Y 587.71,Z 537.437,A -85,B 0,C 180,E1 -1542.014,E2 -1542.014} C_VEL
LIN {X 0,Y 587.748,Z 525.086,A -85,B 0,C 180,E1 -1542.232,E2 -1542.232} C_VEL
LIN {X 0,Y 587.774,Z 423.144,A -85,B 0,C 180,E1 -1543.483,E2 -1543.483} C_VEL
LIN {X 0,Y 587.495,Z 421.014,A -85,B 0,C 180,E1 -1543.534,E2 -1543.534} C_VEL
LIN {X 0,Y 587.64,Z 394.034,A -85,B 0,C 180,E1 -1546.502,E2 -1546.502} C_VEL
LIN {X 0,Y 587.853,Z 368.933,A -85,B 0,C 180,E1 -1549.3,E2 -1549.3} C_VEL
LIN {X 0,Y 588.07,Z 342.491,A -85,B 0,C 180,E1 -1552.299,E2 -1552.299} C_VEL
LIN {X 0,Y 588.282,Z 318.333,A -85,B 0,C 180,E1 -1555.094,E2 -1555.094} C_VEL
LIN {X 0,Y 588.154,Z 311.869,A -85,B 0,C 180,E1 -1555.858,E2 -1555.858} C_VEL
LIN {X 0,Y 587.344,Z 308.327,A -85,B 0,C 180,E1 -1556.302,E2 -1556.302} C_VEL
LIN {X 0,Y 587.346,Z 308.318,A -85,B 0,C 180,E1 -1559.38,E2 -1559.38} C_VEL
LIN {X 0,Y 587.346,Z 308.32,A -85,B 0,C 180,E1 -1561.835,E2 -1561.835} C_VEL
LIN {X 0,Y 587.339,Z 308.328,A -85,B 0,C 180,E1 -1564.346,E2 -1564.346} C_VEL
LIN {X 0,Y 587.343,Z 308.319,A -85,B 0,C 180,E1 -1567.608,E2 -1567.608} C_VEL
LIN {X 0,Y 587.308,Z 308.332,A -85,B 0,C 180,E1 -1570.255,E2 -1570.255} C_VEL
LIN {X 0,Y 587.29,Z 308.325,A -85,B 0,C 180,E1 -1573.009,E2 -1573.009} C_VEL
LIN {X 0,Y 587.306,Z 308.329,A -85,B 0,C 180,E1 -1575.889,E2 -1575.889} C_VEL
LIN {X 0,Y 587.315,Z 308.329,A -85,B 0,C 180,E1 -1577.924,E2 -1577.924} C_VEL
LIN {X 0,Y 587.321,Z 308.322,A -85,B 0,C 180,E1 -1580.638,E2 -1580.638} C_VEL
LIN {X 0,Y 587.31,Z 308.323,A -85,B 0,C 180,E1 -1583.298,E2 -1583.298} C_VEL
LIN {X 0,Y 587.321,Z 308.328,A -85,B 0,C 180,E1 -1585.777,E2 -1585.777} C_VEL
LIN {X 0,Y 587.318,Z 308.325,A -85,B 0,C 180,E1 -1588.229,E2 -1588.229} C_VEL
LIN {X 0,Y 587.3,Z 308.323,A -85,B 0,C 180,E1 -1590.876,E2 -1590.876} C_VEL
LIN {X 0,Y 587.295,Z 308.332,A -85,B 0,C 180,E1 -1593.832,E2 -1593.832} C_VEL
LIN {X 0,Y 587.298,Z 308.324,A -85,B 0,C 180,E1 -1596.74,E2 -1596.74} C_VEL
LIN {X 0,Y 587.301,Z 308.332,A -85,B 0,C 180,E1 -1599.694,E2 -1599.694} C_VEL
LIN {X 0,Y 587.273,Z 308.331,A -85,B 0,C 180,E1 -1601.871,E2 -1601.871} C_VEL
LIN {X 0,Y 587.291,Z 308.327,A -85,B 0,C 180,E1 -1604.024,E2 -1604.024} C_VEL
LIN {X 0,Y 587.325,Z 308.322,A -85,B 0,C 180,E1 -1606.153,E2 -1606.153} C_VEL
LIN {X 0,Y 587.314,Z 308.324,A -85,B 0,C 180,E1 -1608.734,E2 -1608.734} C_VEL
LIN {X 0,Y 587.827,Z 310.715,A -85,B 0,C 180,E1 -1608.779,E2 -1608.779} C_VEL
LIN {X 0,Y 587.682,Z 401.26,A -85,B 0,C 180,E1 -1609.905,E2 -1609.905} C_VEL
LIN {X 0,Y 587.616,Z 414.379,A -85,B 0,C 180,E1 -1610.208,E2 -1610.208} C_VEL
LIN {X 0,Y 587.569,Z 427.506,A -85,B 0,C 180,E1 -1610.664,E2 -1610.664} C_VEL
LIN {X 0,Y 587.547,Z 439.327,A -85,B 0,C 180,E1 -1611.227,E2 -1611.227} C_VEL
LIN {X 0,Y 587.454,Z 449.434,A -85,B 0,C 180,E1 -1611.832,E2 -1611.832} C_VEL
LIN {X 0,Y 587.416,Z 459.935,A -85,B 0,C 180,E1 -1612.61,E2 -1612.61} C_VEL
LIN {X 0,Y 587.339,Z 470.086,A -85,B 0,C 180,E1 -1613.541,E2 -1613.541} C_VEL
LIN {X 0,Y 587.234,Z 478.532,A -85,B 0,C 180,E1 -1614.506,E2 -1614.506} C_VEL
LIN {X 0,Y 587.214,Z 485.866,A -85,B 0,C 180,E1 -1615.538,E2 -1615.538} C_VEL
LIN {X 0,Y 587.201,Z 491.752,A -85,B 0,C 180,E1 -1616.569,E2 -1616.569} C_VEL
LIN {X 0,Y 587.19,Z 496.412,A -85,B 0,C 180,E1 -1617.599,E2 -1617.599} C_VEL
LIN {X 0,Y 587.155,Z 499.984,A -85,B 0,C 180,E1 -1618.628,E2 -1618.628} C_VEL
LIN {X 0,Y 587.141,Z 501.816,A -85,B 0,C 180,E1 -1619.314,E2 -1619.314} C_VEL
LIN {X 0,Y 587.137,Z 503.226,A -85,B 0,C 180,E1 -1620,E2 -1620} C_VEL
LIN {X 0,Y 587.146,Z 504.789,A -85,B 0,C 180,E1 -1621.371,E2 -1621.371} C_VEL
LIN {X 0,Y 587.138,Z 505,A -85,B 0,C 180,E1 -1622.058,E2 -1622.058} C_VEL
LIN {X 0,Y 587.181,Z 504.165,A -85,B 0,C 180,E1 -1623.431,E2 -1623.431} C_VEL
LIN {X 0,Y 587.171,Z 503.18,A -85,B 0,C 180,E1 -1624.118,E2 -1624.118} C_VEL
LIN {X 0,Y 587.132,Z 501.749,A -85,B 0,C 180,E1 -1624.806,E2 -1624.806} C_VEL
LIN {X 0,Y 587.178,Z 498.81,A -85,B 0,C 180,E1 -1625.839,E2 -1625.839} C_VEL
LIN {X 0,Y 587.209,Z 494.834,A -85,B 0,C 180,E1 -1626.874,E2 -1626.874} C_VEL
LIN {X 0,Y 587.217,Z 488.722,A -85,B 0,C 180,E1 -1628.084,E2 -1628.084} C_VEL
LIN {X 0,Y 587.259,Z 482.007,A -85,B 0,C 180,E1 -1629.123,E2 -1629.123} C_VEL
LIN {X 0,Y 587.3,Z 473.619,A -85,B 0,C 180,E1 -1630.166,E2 -1630.166} C_VEL
LIN {X 0,Y 587.364,Z 463.915,A -85,B 0,C 180,E1 -1631.139,E2 -1631.139} C_VEL
LIN {X 0,Y 587.423,Z 453.271,A -85,B 0,C 180,E1 -1631.998,E2 -1631.998} C_VEL
LIN {X 0,Y 587.482,Z 442.322,A -85,B 0,C 180,E1 -1632.698,E2 -1632.698} C_VEL
LIN {X 0,Y 587.606,Z 432.073,A -85,B 0,C 180,E1 -1633.223,E2 -1633.223} C_VEL
LIN {X 0,Y 587.665,Z 421.166,A -85,B 0,C 180,E1 -1633.662,E2 -1633.662} C_VEL
LIN {X 0,Y 587.704,Z 409.156,A -85,B 0,C 180,E1 -1634.017,E2 -1634.017} C_VEL
LIN {X 0,Y 587.728,Z 406.11,A -85,B 0,C 180,E1 -1634.09,E2 -1634.09} C_VEL
LIN {X 0,Y 587.158,Z 400.375,A -85,B 0,C 180,E1 -1634.214,E2 -1634.214} C_VEL
LIN {X 0,Y 581.478,Z 381.737,A -85,B 0,C 180,E1 -1634.58,E2 -1634.58} C_VEL
LIN {X 0,Y 580.816,Z 375.924,A -85,B 0,C 180,E1 -1634.663,E2 -1634.663} C_VEL
LIN {X 0,Y 580.873,Z 311.25,A -85,B 0,C 180,E1 -1635.466,E2 -1635.466} C_VEL
LIN {X 0,Y 580.3,Z 309.197,A -85,B 0,C 180,E1 -1635.52,E2 -1635.52} C_VEL
LIN {X 0,Y 580.29,Z 309.197,A -85,B 0,C 180,E1 -1637.624,E2 -1637.624} C_VEL
LIN {X 0,Y 580.287,Z 309.197,A -85,B 0,C 180,E1 -1639.823,E2 -1639.823} C_VEL
LIN {X 0,Y 580.269,Z 309.2,A -85,B 0,C 180,E1 -1642.052,E2 -1642.052} C_VEL
LIN {X 0,Y 580.305,Z 309.197,A -85,B 0,C 180,E1 -1645.079,E2 -1645.079} C_VEL
LIN {X 0,Y 580.297,Z 309.199,A -85,B 0,C 180,E1 -1648.185,E2 -1648.185} C_VEL
LIN {X 0,Y 580.277,Z 309.206,A -85,B 0,C 180,E1 -1650.693,E2 -1650.693} C_VEL
LIN {X 0,Y 580.284,Z 309.197,A -85,B 0,C 180,E1 -1653.313,E2 -1653.313} C_VEL
LIN {X 0,Y 580.245,Z 309.202,A -85,B 0,C 180,E1 -1655.756,E2 -1655.756} C_VEL
LIN {X 0,Y 580.285,Z 309.201,A -85,B 0,C 180,E1 -1658.146,E2 -1658.146} C_VEL
LIN {X 0,Y 580.297,Z 309.2,A -85,B 0,C 180,E1 -1660.843,E2 -1660.843} C_VEL
LIN {X 0,Y 580.279,Z 309.198,A -85,B 0,C 180,E1 -1663.657,E2 -1663.657} C_VEL
LIN {X 0,Y 580.272,Z 309.205,A -85,B 0,C 180,E1 -1666.609,E2 -1666.609} C_VEL
LIN {X 0,Y 580.297,Z 309.196,A -85,B 0,C 180,E1 -1669.156,E2 -1669.156} C_VEL
LIN {X 0,Y 580.287,Z 309.199,A -85,B 0,C 180,E1 -1671.927,E2 -1671.927} C_VEL
LIN {X 0,Y 580.299,Z 309.204,A -85,B 0,C 180,E1 -1674.456,E2 -1674.456} C_VEL
LIN {X 0,Y 580.289,Z 309.197,A -85,B 0,C 180,E1 -1676.975,E2 -1676.975} C_VEL
LIN {X 0,Y 580.3,Z 309.195,A -85,B 0,C 180,E1 -1679.425,E2 -1679.425} C_VEL
LIN {X 0,Y 580.297,Z 309.203,A -85,B 0,C 180,E1 -1682.141,E2 -1682.141} C_VEL
LIN {X 0,Y 580.32,Z 309.192,A -85,B 0,C 180,E1 -1685.269,E2 -1685.269} C_VEL
LIN {X 0,Y 580.268,Z 309.204,A -85,B 0,C 180,E1 -1687.947,E2 -1687.947} C_VEL
LIN {X 0,Y 580.298,Z 309.196,A -85,B 0,C 180,E1 -1690.913,E2 -1690.913} C_VEL
LIN {X 0,Y 580.306,Z 309.194,A -85,B 0,C 180,E1 -1693.103,E2 -1693.103} C_VEL
LIN {X 0,Y 580.325,Z 309.199,A -85,B 0,C 180,E1 -1695.983,E2 -1695.983} C_VEL
LIN {X 0,Y 580.302,Z 309.195,A -85,B 0,C 180,E1 -1698.827,E2 -1698.827} C_VEL
LIN {X 0,Y 580.326,Z 309.195,A -85,B 0,C 180,E1 -1701.644,E2 -1701.644} C_VEL
LIN {X 0,Y 580.323,Z 309.196,A -85,B 0,C 180,E1 -1704.44,E2 -1704.44} C_VEL
LIN {X 0,Y 580.335,Z 309.191,A -85,B 0,C 180,E1 -1707.224,E2 -1707.224} C_VEL
LIN {X 0,Y 580.352,Z 309.198,A -85,B 0,C 180,E1 -1710,E2 -1710} C_VEL
LIN {X 0,Y 580.335,Z 309.191,A -85,B 0,C 180,E1 -1712.777,E2 -1712.777} C_VEL
LIN {X 0,Y 580.323,Z 309.196,A -85,B 0,C 180,E1 -1715.56,E2 -1715.56} C_VEL
LIN {X 0,Y 580.326,Z 309.195,A -85,B 0,C 180,E1 -1718.356,E2 -1718.356} C_VEL
LIN {X 0,Y 580.298,Z 309.196,A -85,B 0,C 180,E1 -1721.191,E2 -1721.191} C_VEL
LIN {X 0,Y 580.325,Z 309.2,A -85,B 0,C 180,E1 -1724.017,E2 -1724.017} C_VEL
LIN {X 0,Y 580.311,Z 309.193,A -85,B 0,C 180,E1 -1726.914,E2 -1726.914} C_VEL
LIN {X 0,Y 580.302,Z 309.204,A -85,B 0,C 180,E1 -1729.823,E2 -1729.823} C_VEL
LIN {X 0,Y 580.294,Z 309.195,A -85,B 0,C 180,E1 -1732.803,E2 -1732.803} C_VEL
LIN {X 0,Y 580.307,Z 309.195,A -85,B 0,C 180,E1 -1735.08,E2 -1735.08} C_VEL
LIN {X 0,Y 580.299,Z 309.198,A -85,B 0,C 180,E1 -1738.186,E2 -1738.186} C_VEL
LIN {X 0,Y 580.292,Z 309.196,A -85,B 0,C 180,E1 -1740.696,E2 -1740.696} C_VEL
LIN {X 0,Y 580.303,Z 309.199,A -85,B 0,C 180,E1 -1743.317,E2 -1743.317} C_VEL
LIN {X 0,Y 580.272,Z 309.207,A -85,B 0,C 180,E1 -1745.76,E2 -1745.76} C_VEL
LIN {X 0,Y 580.287,Z 309.199,A -85,B 0,C 180,E1 -1748.147,E2 -1748.147} C_VEL
LIN {X 0,Y 580.298,Z 309.195,A -85,B 0,C 180,E1 -1750.844,E2 -1750.844} C_VEL
LIN {X 0,Y 580.273,Z 309.208,A -85,B 0,C 180,E1 -1753.659,E2 -1753.659} C_VEL
LIN {X 0,Y 580.279,Z 309.197,A -85,B 0,C 180,E1 -1756.61,E2 -1756.61} C_VEL
LIN {X 0,Y 580.298,Z 309.199,A -85,B 0,C 180,E1 -1759.157,E2 -1759.157} C_VEL
LIN {X 0,Y 580.289,Z 309.2,A -85,B 0,C 180,E1 -1761.928,E2 -1761.928} C_VEL
LIN {X 0,Y 580.252,Z 309.201,A -85,B 0,C 180,E1 -1764.453,E2 -1764.453} C_VEL
LIN {X 0,Y 580.291,Z 309.199,A -85,B 0,C 180,E1 -1766.976,E2 -1766.976} C_VEL
LIN {X 0,Y 580.289,Z 309.206,A -85,B 0,C 180,E1 -1769.425,E2 -1769.425} C_VEL
LIN {X 0,Y 580.294,Z 309.196,A -85,B 0,C 180,E1 -1772.143,E2 -1772.143} C_VEL
LIN {X 0,Y 580.324,Z 309.2,A -85,B 0,C 180,E1 -1775.271,E2 -1775.271} C_VEL
LIN {X 0,Y 580.283,Z 309.198,A -85,B 0,C 180,E1 -1778.322,E2 -1778.322} C_VEL
LIN {X 0,Y 580.309,Z 309.196,A -85,B 0,C 180,E1 -1778.57,E2 -1778.57} C_VEL
LIN {X 0,Y 580.955,Z 312.154,A -85,B 0,C 180,E1 -1778.637,E2 -1778.637} C_VEL
LIN {X 0,Y 580.783,Z 400.943,A -85,B 0,C 180,E1 -1779.757,E2 -1779.757} C_VEL
LIN {X 0,Y 580.737,Z 413.195,A -85,B 0,C 180,E1 -1780.032,E2 -1780.032} C_VEL
LIN {X 0,Y 580.624,Z 427.401,A -85,B 0,C 180,E1 -1780.522,E2 -1780.522} C_VEL
LIN {X 0,Y 580.562,Z 439.5,A -85,B 0,C 180,E1 -1781.106,E2 -1781.106} C_VEL
LIN {X 0,Y 580.45,Z 449.942,A -85,B 0,C 180,E1 -1781.743,E2 -1781.743} C_VEL
LIN {X 0,Y 580.392,Z 459.639,A -85,B 0,C 180,E1 -1782.47,E2 -1782.47} C_VEL
LIN {X 0,Y 580.271,Z 468.56,A -85,B 0,C 180,E1 -1783.283,E2 -1783.283} C_VEL
LIN {X 0,Y 580.232,Z 478.155,A -85,B 0,C 180,E1 -1784.366,E2 -1784.366} C_VEL
LIN {X 0,Y 580.166,Z 484.616,A -85,B 0,C 180,E1 -1785.263,E2 -1785.263} C_VEL
LIN {X 0,Y 580.115,Z 490.895,A -85,B 0,C 180,E1 -1786.336,E2 -1786.336} C_VEL
LIN {X 0,Y 580.097,Z 495.835,A -85,B 0,C 180,E1 -1787.404,E2 -1787.404} C_VEL
LIN {X 0,Y 580.076,Z 499.622,A -85,B 0,C 180,E1 -1788.469,E2 -1788.469} C_VEL
LIN {X 0,Y 580.059,Z 502.351,A -85,B 0,C 180,E1 -1789.529,E2 -1789.529} C_VEL
LIN {X 0,Y 580.057,Z 503.635,A -85,B 0,C 180,E1 -1790.234,E2 -1790.234} C_VEL
LIN {X 0,Y 580.027,Z 504.495,A -85,B 0,C 180,E1 -1790.938,E2 -1790.938} C_VEL
LIN {X 0,Y 580.067,Z 504.94,A -85,B 0,C 180,E1 -1792.342,E2 -1792.342} C_VEL
LIN {X 0,Y 580.101,Z 504.176,A -85,B 0,C 180,E1 -1793.438,E2 -1793.438} C_VEL
LIN {X 0,Y 580.099,Z 502.607,A -85,B 0,C 180,E1 -1794.438,E2 -1794.438} C_VEL
LIN {X 0,Y 580.103,Z 500.041,A -85,B 0,C 180,E1 -1795.484,E2 -1795.484} C_VEL
LIN {X 0,Y 580.126,Z 496.478,A -85,B 0,C 180,E1 -1796.528,E2 -1796.528} C_VEL
LIN {X 0,Y 580.112,Z 491.836,A -85,B 0,C 180,E1 -1797.57,E2 -1797.57} C_VEL
LIN {X 0,Y 580.121,Z 485.978,A -85,B 0,C 180,E1 -1798.612,E2 -1798.612} C_VEL
LIN {X 0,Y 580.204,Z 478.708,A -85,B 0,C 180,E1 -1799.653,E2 -1799.653} C_VEL
LIN {X 0,Y 580.273,Z 469.694,A -85,B 0,C 180,E1 -1800.694,E2 -1800.694} C_VEL
LIN {X 0,Y 580.376,Z 459.291,A -85,B 0,C 180,E1 -1801.648,E2 -1801.648} C_VEL
LIN {X 0,Y 580.426,Z 450.021,A -85,B 0,C 180,E1 -1802.342,E2 -1802.342} C_VEL
LIN {X 0,Y 580.54,Z 440.125,A -85,B 0,C 180,E1 -1802.95,E2 -1802.95} C_VEL
LIN {X 0,Y 580.6,Z 429.592,A -85,B 0,C 180,E1 -1803.47,E2 -1803.47} C_VEL
LIN {X 0,Y 580.662,Z 418.256,A -85,B 0,C 180,E1 -1803.904,E2 -1803.904} C_VEL
LIN {X 0,Y 580.732,Z 405.459,A -85,B 0,C 180,E1 -1804.251,E2 -1804.251} C_VEL
LIN {X 0,Y 580.777,Z 388.207,A -85,B 0,C 180,E1 -1804.512,E2 -1804.512} C_VEL
LIN {X 0,Y 580.813,Z 311.172,A -85,B 0,C 180,E1 -1805.468,E2 -1805.468} C_VEL
LIN {X 0,Y 580.283,Z 309.199,A -85,B 0,C 180,E1 -1805.517,E2 -1805.517} C_VEL
LIN {X 0,Y 580.291,Z 309.202,A -85,B 0,C 180,E1 -1808.357,E2 -1808.357} C_VEL
LIN {X 0,Y 580.273,Z 309.201,A -85,B 0,C 180,E1 -1811.174,E2 -1811.174} C_VEL
LIN {X 0,Y 580.291,Z 309.199,A -85,B 0,C 180,E1 -1814.018,E2 -1814.018} C_VEL
LIN {X 0,Y 580.273,Z 309.202,A -85,B 0,C 180,E1 -1816.899,E2 -1816.899} C_VEL
LIN {X 0,Y 580.249,Z 309.204,A -85,B 0,C 180,E1 -1819.825,E2 -1819.825} C_VEL
LIN {X 0,Y 580.283,Z 309.2,A -85,B 0,C 180,E1 -1822.803,E2 -1822.803} C_VEL
LIN {X 0,Y 580.241,Z 309.203,A -85,B 0,C 180,E1 -1825.083,E2 -1825.083} C_VEL
LIN {X 0,Y 580.239,Z 309.207,A -85,B 0,C 180,E1 -1827.846,E2 -1827.846} C_VEL
LIN {X 0,Y 580.262,Z 309.202,A -85,B 0,C 180,E1 -1830.69,E2 -1830.69} C_VEL
LIN {X 0,Y 580.282,Z 309.198,A -85,B 0,C 180,E1 -1833.312,E2 -1833.312} C_VEL
LIN {X 0,Y 580.226,Z 309.209,A -85,B 0,C 180,E1 -1835.753,E2 -1835.753} C_VEL
LIN {X 0,Y 580.282,Z 309.204,A -85,B 0,C 180,E1 -1838.147,E2 -1838.147} C_VEL
LIN {X 0,Y 580.279,Z 309.197,A -85,B 0,C 180,E1 -1840.845,E2 -1840.845} C_VEL
LIN {X 0,Y 580.241,Z 309.208,A -85,B 0,C 180,E1 -1843.662,E2 -1843.662} C_VEL
LIN {X 0,Y 580.238,Z 309.203,A -85,B 0,C 180,E1 -1846.614,E2 -1846.614} C_VEL
LIN {X 0,Y 580.283,Z 309.199,A -85,B 0,C 180,E1 -1849.155,E2 -1849.155} C_VEL
LIN {X 0,Y 580.286,Z 309.203,A -85,B 0,C 180,E1 -1851.928,E2 -1851.928} C_VEL
LIN {X 0,Y 580.236,Z 309.203,A -85,B 0,C 180,E1 -1854.451,E2 -1854.451} C_VEL
LIN {X 0,Y 580.292,Z 309.198,A -85,B 0,C 180,E1 -1856.975,E2 -1856.975} C_VEL
LIN {X 0,Y 580.296,Z 309.204,A -85,B 0,C 180,E1 -1859.425,E2 -1859.425} C_VEL
LIN {X 0,Y 580.262,Z 309.203,A -85,B 0,C 180,E1 -1862.149,E2 -1862.149} C_VEL
LIN {X 0,Y 580.292,Z 309.246,A -85,B 0,C 180,E1 -1863.536,E2 -1863.536} C_VEL
LIN {X 0,Y 581.435,Z 314.669,A -85,B 0,C 180,E1 -1864.205,E2 -1864.205} C_VEL
LIN {X 0,Y 581.321,Z 335.614,A -85,B 0,C 180,E1 -1866.625,E2 -1866.625} C_VEL
LIN {X 0,Y 581.037,Z 360.207,A -85,B 0,C 180,E1 -1869.465,E2 -1869.465} C_VEL
LIN {X 0,Y 580.788,Z 385.978,A -85,B 0,C 180,E1 -1872.391,E2 -1872.391} C_VEL
LIN {X 0,Y 580.55,Z 411.75,A -85,B 0,C 180,E1 -1875.272,E2 -1875.272} C_VEL
LIN {X 0,Y 580.511,Z 421.336,A -85,B 0,C 180,E1 -1876.322,E2 -1876.322} C_VEL
LIN {X 0,Y 580.968,Z 426.702,A -85,B 0,C 180,E1 -1876.4,E2 -1876.4} C_VEL
LIN {X 0,Y 580.771,Z 530.936,A -85,B 0,C 180,E1 -1877.707,E2 -1877.707} C_VEL
LIN {X 0,Y 580.727,Z 544.212,A -85,B 0,C 180,E1 -1878.017,E2 -1878.017} C_VEL
LIN {X 0,Y 580.629,Z 556.368,A -85,B 0,C 180,E1 -1878.435,E2 -1878.435} C_VEL
LIN {X 0,Y 580.567,Z 568.626,A -85,B 0,C 180,E1 -1879.009,E2 -1879.009} C_VEL
LIN {X 0,Y 580.444,Z 580.2,A -85,B 0,C 180,E1 -1879.712,E2 -1879.712} C_VEL
LIN {X 0,Y 580.341,Z 590.597,A -85,B 0,C 180,E1 -1880.503,E2 -1880.503} C_VEL
LIN {X 0,Y 580.272,Z 599.111,A -85,B 0,C 180,E1 -1881.292,E2 -1881.292} C_VEL
LIN {X 0,Y 580.222,Z 606.959,A -85,B 0,C 180,E1 -1882.168,E2 -1882.168} C_VEL
LIN {X 0,Y 580.154,Z 614.65,A -85,B 0,C 180,E1 -1883.222,E2 -1883.222} C_VEL
LIN {X 0,Y 580.139,Z 621.679,A -85,B 0,C 180,E1 -1884.438,E2 -1884.438} C_VEL
LIN {X 0,Y 580.108,Z 626.371,A -85,B 0,C 180,E1 -1885.483,E2 -1885.483} C_VEL
LIN {X 0,Y 580.123,Z 629.956,A -85,B 0,C 180,E1 -1886.527,E2 -1886.527} C_VEL
LIN {X 0,Y 580.043,Z 631.808,A -85,B 0,C 180,E1 -1887.222,E2 -1887.222} C_VEL
LIN {X 0,Y 580.038,Z 633.199,A -85,B 0,C 180,E1 -1887.917,E2 -1887.917} C_VEL
LIN {X 0,Y 580.04,Z 634.785,A -85,B 0,C 180,E1 -1889.306,E2 -1889.306} C_VEL
LIN {X 0,Y 580.037,Z 635,A -85,B 0,C 180,E1 -1890,E2 -1890} C_VEL
LIN {X 0,Y 580.047,Z 634.186,A -85,B 0,C 180,E1 -1891.388,E2 -1891.388} C_VEL
LIN {X 0,Y 580.038,Z 633.2,A -85,B 0,C 180,E1 -1892.083,E2 -1892.083} C_VEL
LIN {X 0,Y 580.043,Z 631.81,A -85,B 0,C 180,E1 -1892.778,E2 -1892.778} C_VEL
LIN {X 0,Y 580.109,Z 628.896,A -85,B 0,C 180,E1 -1893.82,E2 -1893.82} C_VEL
LIN {X 0,Y 580.054,Z 624.95,A -85,B 0,C 180,E1 -1894.865,E2 -1894.865} C_VEL
LIN {X 0,Y 580.139,Z 618.878,A -85,B 0,C 180,E1 -1896.085,E2 -1896.085} C_VEL
LIN {X 0,Y 580.184,Z 612.238,A -85,B 0,C 180,E1 -1897.132,E2 -1897.132} C_VEL
LIN {X 0,Y 580.25,Z 603.991,A -85,B 0,C 180,E1 -1898.182,E2 -1898.182} C_VEL
LIN {X 0,Y 580.308,Z 595.539,A -85,B 0,C 180,E1 -1899.058,E2 -1899.058} C_VEL
LIN {X 0,Y 580.417,Z 585.097,A -85,B 0,C 180,E1 -1899.936,E2 -1899.936} C_VEL
LIN {X 0,Y 580.507,Z 574.757,A -85,B 0,C 180,E1 -1900.639,E2 -1900.639} C_VEL
LIN {X 0,Y 580.597,Z 563.24,A -85,B 0,C 180,E1 -1901.264,E2 -1901.264} C_VEL
LIN {X 0,Y 580.665,Z 550.472,A -85,B 0,C 180,E1 -1901.785,E2 -1901.785} C_VEL
LIN {X 0,Y 580.781,Z 537.436,A -85,B 0,C 180,E1 -1902.159,E2 -1902.159} C_VEL
LIN {X 0,Y 580.82,Z 525.086,A -85,B 0,C 180,E1 -1902.38,E2 -1902.38} C_VEL
LIN {X 0,Y 580.836,Z 423.591,A -85,B 0,C 180,E1 -1903.642,E2 -1903.642} C_VEL
LIN {X 0,Y 580.493,Z 421.014,A -85,B 0,C 180,E1 -1903.7,E2 -1903.7} C_VEL
LIN {X 0,Y 580.702,Z 394.034,A -85,B 0,C 180,E1 -1906.705,E2 -1906.705} C_VEL
LIN {X 0,Y 580.936,Z 369.315,A -85,B 0,C 180,E1 -1909.496,E2 -1909.496} C_VEL
LIN {X 0,Y 581.214,Z 344.101,A -85,B 0,C 180,E1 -1912.389,E2 -1912.389} C_VEL
LIN {X 0,Y 581.454,Z 321.285,A -85,B 0,C 180,E1 -1915.027,E2 -1915.027} C_VEL
LIN {X 0,Y 581.374,Z 314.375,A -85,B 0,C 180,E1 -1915.797,E2 -1915.797} C_VEL
LIN {X 0,Y 580.299,Z 309.205,A -85,B 0,C 180,E1 -1916.421,E2 -1916.421} C_VEL
LIN {X 0,Y 580.301,Z 309.197,A -85,B 0,C 180,E1 -1919.309,E2 -1919.309} C_VEL
LIN {X 0,Y 580.301,Z 309.202,A -85,B 0,C 180,E1 -1922.2,E2 -1922.2} C_VEL
LIN {X 0,Y 580.286,Z 309.202,A -85,B 0,C 180,E1 -1924.697,E2 -1924.697} C_VEL
LIN {X 0,Y 580.29,Z 309.197,A -85,B 0,C 180,E1 -1927.269,E2 -1927.269} C_VEL
LIN {X 0,Y 580.288,Z 309.206,A -85,B 0,C 180,E1 -1930.27,E2 -1930.27} C_VEL
LIN {X 0,Y 580.264,Z 309.202,A -85,B 0,C 180,E1 -1932.708,E2 -1932.708} C_VEL
LIN {X 0,Y 580.253,Z 309.203,A -85,B 0,C 180,E1 -1935.611,E2 -1935.611} C_VEL
LIN {X 0,Y 580.252,Z 309.209,A -85,B 0,C 180,E1 -1938.228,E2 -1938.228} C_VEL
LIN {X 0,Y 580.264,Z 309.199,A -85,B 0,C 180,E1 -1940.964,E2 -1940.964} C_VEL
LIN {X 0,Y 580.24,Z 309.207,A -85,B 0,C 180,E1 -1943.594,E2 -1943.594} C_VEL
LIN {X 0,Y 580.271,Z 309.204,A -85,B 0,C 180,E1 -1946.142,E2 -1946.142} C_VEL
LIN {X 0,Y 580.25,Z 309.202,A -85,B 0,C 180,E1 -1948.613,E2 -1948.613} C_VEL
LIN {X 0,Y 580.247,Z 309.202,A -85,B 0,C 180,E1 -1951.021,E2 -1951.021} C_VEL
LIN {X 0,Y 580.248,Z 309.211,A -85,B 0,C 180,E1 -1953.675,E2 -1953.675} C_VEL
LIN {X 0,Y 580.252,Z 309.202,A -85,B 0,C 180,E1 -1956.441,E2 -1956.441} C_VEL
LIN {X 0,Y 580.245,Z 309.21,A -85,B 0,C 180,E1 -1959.436,E2 -1959.436} C_VEL
LIN {X 0,Y 580.233,Z 309.212,A -85,B 0,C 180,E1 -1961.644,E2 -1961.644} C_VEL
LIN {X 0,Y 580.246,Z 309.208,A -85,B 0,C 180,E1 -1963.824,E2 -1963.824} C_VEL
LIN {X 0,Y 580.291,Z 309.2,A -85,B 0,C 180,E1 -1965.982,E2 -1965.982} C_VEL
LIN {X 0,Y 580.263,Z 309.202,A -85,B 0,C 180,E1 -1968.584,E2 -1968.584} C_VEL
LIN {X 0,Y 580.928,Z 312.76,A -85,B 0,C 180,E1 -1968.644,E2 -1968.644} C_VEL
LIN {X 0,Y 580.761,Z 401.43,A -85,B 0,C 180,E1 -1969.762,E2 -1969.762} C_VEL
LIN {X 0,Y 580.688,Z 414.497,A -85,B 0,C 180,E1 -1970.068,E2 -1970.068} C_VEL
LIN {X 0,Y 580.617,Z 427.06,A -85,B 0,C 180,E1 -1970.507,E2 -1970.507} C_VEL
LIN {X 0,Y 580.578,Z 438.197,A -85,B 0,C 180,E1 -1971.033,E2 -1971.033} C_VEL
LIN {X 0,Y 580.461,Z 448.497,A -85,B 0,C 180,E1 -1971.646,E2 -1971.646} C_VEL
LIN {X 0,Y 580.381,Z 458.085,A -85,B 0,C 180,E1 -1972.345,E2 -1972.345} C_VEL
LIN {X 0,Y 580.298,Z 467.318,A -85,B 0,C 180,E1 -1973.162,E2 -1973.162} C_VEL
LIN {X 0,Y 580.214,Z 475.921,A -85,B 0,C 180,E1 -1974.09,E2 -1974.09} C_VEL
LIN {X 0,Y 580.224,Z 483.797,A -85,B 0,C 180,E1 -1975.136,E2 -1975.136} C_VEL
LIN {X 0,Y 580.148,Z 490.083,A -85,B 0,C 180,E1 -1976.179,E2 -1976.179} C_VEL
LIN {X 0,Y 580.066,Z 495.094,A -85,B 0,C 180,E1 -1977.222,E2 -1977.222} C_VEL
LIN {X 0,Y 580.086,Z 498.986,A -85,B 0,C 180,E1 -1978.264,E2 -1978.264} C_VEL
LIN {X 0,Y 580.042,Z 501.862,A -85,B 0,C 180,E1 -1979.305,E2 -1979.305} C_VEL
LIN {X 0,Y 580.038,Z 503.267,A -85,B 0,C 180,E1 -1980,E2 -1980} C_VEL
LIN {X 0,Y 580.046,Z 504.791,A -85,B 0,C 180,E1 -1981.388,E2 -1981.388} C_VEL
LIN {X 0,Y 580.037,Z 504.997,A -85,B 0,C 180,E1 -1982.083,E2 -1982.083} C_VEL
LIN {X 0,Y 580.106,Z 504.133,A -85,B 0,C 180,E1 -1983.472,E2 -1983.472} C_VEL
LIN {X 0,Y 580.088,Z 503.141,A -85,B 0,C 180,E1 -1984.168,E2 -1984.168} C_VEL
LIN {X 0,Y 580.036,Z 501.685,A -85,B 0,C 180,E1 -1984.865,E2 -1984.865} C_VEL
LIN {X 0,Y 580.093,Z 498.724,A -85,B 0,C 180,E1 -1985.91,E2 -1985.91} C_VEL
LIN {X 0,Y 580.14,Z 494.725,A -85,B 0,C 180,E1 -1986.958,E2 -1986.958} C_VEL
LIN {X 0,Y 580.153,Z 488.578,A -85,B 0,C 180,E1 -1988.183,E2 -1988.183} C_VEL
LIN {X 0,Y 580.204,Z 481.828,A -85,B 0,C 180,E1 -1989.235,E2 -1989.235} C_VEL
LIN {X 0,Y 580.268,Z 473.381,A -85,B 0,C 180,E1 -1990.291,E2 -1990.291} C_VEL
LIN {X 0,Y 580.311,Z 464.524,A -85,B 0,C 180,E1 -1991.194,E2 -1991.194} C_VEL
LIN {X 0,Y 580.395,Z 454.114,A -85,B 0,C 180,E1 -1992.056,E2 -1992.056} C_VEL
LIN {X 0,Y 580.476,Z 443.433,A -85,B 0,C 180,E1 -1992.765,E2 -1992.765} C_VEL
LIN {X 0,Y 580.615,Z 433.457,A -85,B 0,C 180,E1 -1993.296,E2 -1993.296} C_VEL
LIN {X 0,Y 580.713,Z 421.674,A -85,B 0,C 180,E1 -1993.784,E2 -1993.784} C_VEL
LIN {X 0,Y 580.723,Z 409.92,A -85,B 0,C 180,E1 -1994.143,E2 -1994.143} C_VEL
LIN {X 0,Y 580.834,Z 397.702,A -85,B 0,C 180,E1 -1994.387,E2 -1994.387} C_VEL
LIN {X 0,Y 580.816,Z 375.924,A -85,B 0,C 180,E1 -1994.663,E2 -1994.663} C_VEL
LIN {X 0,Y 580.182,Z 370.117,A -85,B 0,C 180,E1 -1994.749,E2 -1994.749} C_VEL
LIN {X 0,Y 574.638,Z 351.421,A -85,B 0,C 180,E1 -1995.109,E2 -1995.109} C_VEL
LIN {X 0,Y 573.988,Z 345.614,A -85,B 0,C 180,E1 -1995.197,E2 -1995.197} C_VEL
LIN {X 0,Y 573.88,Z 312.294,A -85,B 0,C 180,E1 -1995.619,E2 -1995.619} C_VEL
LIN {X 0,Y 573.269,Z 310.073,A -85,B 0,C 180,E1 -1995.669,E2 -1995.669} C_VEL
LIN {X 0,Y 573.241,Z 310.075,A -85,B 0,C 180,E1 -1997.848,E2 -1997.848} C_VEL
LIN {X 0,Y 573.242,Z 310.076,A -85,B 0,C 180,E1 -2000.077,E2 -2000.077} C_VEL
LIN {X 0,Y 573.234,Z 310.08,A -85,B 0,C 180,E1 -2002.338,E2 -2002.338} C_VEL
LIN {X 0,Y 573.249,Z 310.074,A -85,B 0,C 180,E1 -2005.41,E2 -2005.41} C_VEL
